# B&R Automation Studio project GAT (part 4)

#### AlarmMgt.st
```iecst
//***********************************************************************
// Copyright: B&R Industrial Automation GmbH
// Author: B&R Industrial Automation GmbH
// Created: Jan 1, 2022
// Description: Tasks for alarm control. The Alarm Management handling is
// done in this task.
//***********************************************************************

PROGRAM _INIT

	// Create folder for this component on the user file device
	DirCreate_New(enable := TRUE, pDevice := ADR('userPartition'), pName := ADR(LOCAL_FOLDER));

	// Check if folder already exist and if so disabled the function block call
	IF DirCreate_New.status = fiERR_DIR_ALREADY_EXIST THEN
		DirCreate_New(enable := FALSE);
	END_IF

	// Initialize mapp function blocks
	MpAlarmXCore_0.Enable := TRUE;
	MpAlarmXCore_0.MpLink := ADR(gMpLinkAlarmXCore);
	MpAlarmXCore_0();

	MpAlarmXHistory_0.Enable := TRUE;
	MpAlarmXHistory_0.DeviceName := ADR('mappAlarmX');
	MpAlarmXHistory_0.MpLink := ADR(gMpLinkAlarmXHistory);
	MpAlarmXHistory_0();

	MpAlarmXListUI_0.Enable := TRUE;
	MpAlarmXListUI_0.UISetup.AlarmListScrollWindow := 10;
	MpAlarmXListUI_0.UISetup.AlarmListSize := 50;
	MpAlarmXListUI_0.UISetup.TimeStampPattern := '%Y %m %d %H:%M:%S';
	MpAlarmXListUI_0();

	MpAlarmXHistoryUI_0.Enable := TRUE;
	MpAlarmXHistoryUI_0.UISetup.AlarmListScrollWindow := 10;
    MpAlarmXHistoryUI_0.UISetup.AlarmListSize := (SIZEOF(MpAlarmXListUIConnect.AlarmList.InstanceID) / SIZEOF(MpAlarmXListUIConnect.AlarmList.InstanceID[0]));
	MpAlarmXHistoryUI_0.UISetup.TimeStampPattern := '%Y %m %d %H:%M:%S';
	MpAlarmXHistoryUI_0();

	// Call action to intialize alarm samples
	AlarmSampleInit;

END_PROGRAM

PROGRAM _CYCLIC

	IF EDGEPOS(SafetyInputs.AcknowledgeAlarms) THEN
        MpAlarmXListUIConnect.AcknowledgeAll := TRUE;
	END_IF

	IF (HmiAlarmX.Commands.ExportAlarms = TRUE) THEN
		MpAlarmXHistory_0.Export := TRUE;
	END_IF

    // Call all cyclic actions
    AlarmHandling;
    GetBacktraceInformation;
    ExecuteQuery;
    QueryTableConfig;
    AlarmSampleFub;

	// Check if any reactions are active.
	// Typically the MpAlarmXCheckReaction() function is called from other tasks within the application.
	// For example, the axis control task might check for the 'Error' reaction to determine whether to send a stop command to the axes.
	// Therefore, copy/paste these IF statements to other places in the application as needed.
    IF MpAlarmXCheckReaction(gMpLinkAlarmXCore, 'Error') THEN
        // Error is active. Add code here to respond to error situation.
    ELSIF MpAlarmXCheckReaction(gMpLinkAlarmXCore, 'Warning') THEN
        // Warning is active. Add code here to respond to warning situation.
	ELSIF MpAlarmXCheckReaction(gMpLinkAlarmXCore, 'Info') THEN
        // Info is active. Add code here to resond to info situation.
	END_IF

	IF ((MpAlarmXHistory_0.Export = TRUE) AND (MpAlarmXHistory_0.CommandDone = TRUE)) THEN
		HmiAlarmX.Commands.ExportAlarms := FALSE;
		MpAlarmXHistory_0.Export := FALSE;
	END_IF

    // Error reset
    IF NOT MpAlarmXCore_0.Error THEN
        MpAlarmXCore_0.ErrorReset := FALSE;
    END_IF
    IF NOT MpAlarmXListUI_0.Error THEN
        MpAlarmXListUI_0.ErrorReset := FALSE;
    END_IF
    IF NOT MpAlarmXHistory_0.Error THEN
        MpAlarmXHistory_0.ErrorReset := FALSE;
    END_IF
    IF NOT MpAlarmXHistoryUI_0.Error THEN
        MpAlarmXHistoryUI_0.ErrorReset := FALSE;
    END_IF

	// Assign MpLinks & UIConnects
	MpAlarmXCore_0.MpLink := ADR(gMpLinkAlarmXCore);
	MpAlarmXListUI_0.MpLink := ADR(gMpLinkAlarmXCore);
	MpAlarmXListUI_0.UIConnect := ADR(MpAlarmXListUIConnect);
	MpAlarmXHistory_0.MpLink := ADR(gMpLinkAlarmXHistory);
	MpAlarmXHistoryUI_0.MpLink := ADR(gMpLinkAlarmXHistory);
	MpAlarmXHistoryUI_0.UIConnect := ADR(MpAlarmXHistoryUIConnect);

	// Call function blocks
	MpAlarmXCore_0();
	MpAlarmXListUI_0();
	MpAlarmXHistory_0();
	MpAlarmXHistoryUI_0();

END_PROGRAM

PROGRAM _EXIT

	// Disable the function blocls to unlink the MpLinks
    MpAlarmXCore_0.Enable := FALSE;
    MpAlarmXListUI_0.Enable := FALSE;
    MpAlarmXHistory_0.Enable := FALSE;
	MpAlarmXHistoryUI_0.Enable := FALSE;
	QueryActiveAlarms.Enable := FALSE;

	// Call function blocks
    MpAlarmXCore_0();
    MpAlarmXListUI_0();
    MpAlarmXHistory_0();
    MpAlarmXHistoryUI_0();
    QueryActiveAlarms();

END_PROGRAM
```

#### AlarmMgt.typ
```iecst
TYPE
	MachineDigitalInputs_type : 	STRUCT  (*Safety related digital inputs of the machine*)
		EmergencyStop : ARRAY[0..MAX_IDX_ESTOP]OF BOOL; (*Emergency stop signal*)
		SafetyDoor : ARRAY[0..MAX_IDX_SAFETY_DOOR]OF BOOL; (*Safety door signal*)
		AcknowledgeAlarms : BOOL;
	END_STRUCT;
	AlarmExamples_typ : 	STRUCT
		LevelMonitoring : INT;
		DeviationMonitoring : INT;
		DeviationMonitoringSetpoint : INT;
		RateOfChange : INT;
		SnippetValue : INT;
		SetControlExample : BOOL;
	END_STRUCT;
	ActiveAlarmState_enum :
		(
		ACTIVE_ALARM_WAIT,
		ACTIVE_ALARM_QUERY,
		ACTIVE_ALARM_NEXT
		);
	AlarmType : 	STRUCT
		Active : BOOL;
		Acknowledged : BOOL;
		Scope : WSTRING[80];
		Name : STRING[80];
		Message : WSTRING[255];
		AdditionalInfo : WSTRING[255];
		TimeStamp : DATE_AND_TIME;
		Code : UDINT;
		Severity : UDINT;
	END_STRUCT;
	AlarmQueryType : 	STRUCT
		Next : BOOL;
		State : ActiveAlarmState_enum;
		LastActiveAlarmUpdateCount : UDINT;
		ActiveAlarmUpdateCount : UDINT;
		Alarms : ARRAY[0..MAX_QUERY_RESULTS]OF AlarmType;
	END_STRUCT;
	AlarmHmiInterface_type : 	STRUCT
		Commands : AlarmCommands_type;
		Status : AlarmStatus_type;
	END_STRUCT;
	AlarmStatus_type : 	STRUCT
		AlarmHistSortCfg : STRING[1000];
		AlarmHistFilterCfg : STRING[1000];
		AlarmSortCfg : STRING[1000];
		AlarmFilterCfg : STRING[1000];
		TableConfig : ARRAY[0..1]OF STRING[120];
	END_STRUCT;
	AlarmCommands_type : 	STRUCT
		ExportAlarms : BOOL;
		RunQuery : BOOL;
	END_STRUCT;
	AlarmQueryHMI_type : 	STRUCT
		Active : ARRAY[0..MAX_QUERY_RESULTS]OF BOOL;
		Acknowledged : ARRAY[0..MAX_QUERY_RESULTS]OF BOOL;
		Scope : ARRAY[0..MAX_QUERY_RESULTS]OF WSTRING[80];
		Name : ARRAY[0..MAX_QUERY_RESULTS]OF STRING[80];
		Message : ARRAY[0..MAX_QUERY_RESULTS]OF WSTRING[255];
		AdditionalInfo : ARRAY[0..MAX_QUERY_RESULTS]OF WSTRING[255];
		TimeStamp : ARRAY[0..MAX_QUERY_RESULTS]OF DATE_AND_TIME;
		Code : ARRAY[0..MAX_QUERY_RESULTS]OF UDINT;
		Severity : ARRAY[0..MAX_QUERY_RESULTS]OF UDINT;
	END_STRUCT;
END_TYPE
```

#### AlarmMgt.var - Local variables
```iecst
(********************************************************************
 * COPYRIGHT -- Bernecker + Rainer
 ********************************************************************
 * Program: FolderHandling
 * File: FolderHandling.var
 * Author: Bernecker + Rainer
 * Created: December , 2020
 ********************************************************************
 * Local variables of program AlarmManagement
 ********************************************************************)
(*Function Blocks--------------------------------------------------------------------------------------------------------------------*)
VAR
	HmiAlarmX : AlarmHmiInterfaceType;
	MpAlarmXHistory_0 : MpAlarmXHistory; (*MpAlarmXHistory instance*)
	MpAlarmXHistoryUI_0 : MpAlarmXHistoryUI; (*MpAlarmXHistoryUI instance*)
	MpAlarmXListUI_0 : MpAlarmXListUI; (*MpAlarmXList instance*)
	MpAlarmXCore_0 : MpAlarmXCore; (*MpAlarmXCore instance*) (*ChangeStyleAlarmButton : USINT := 0; (*changeStyle of a AlarmFlyout in mappView*)
	DirCreate_New : DirCreate;
END_VAR
(*Alarm Management Variables------------------------------------------------------------------------------------------------*)
VAR
	Index : USINT; (*Index to loop through alarm list*)
	MaxIndex : USINT; (*Maximum index for the alarm list*)
	InstanceID : UINT; (*Instance ID*)
	MpAlarmXListUIConnect : MpAlarmXListUIConnectType := (0); (*AlarmVideo : WSTRING[255] := "";
	AlarmInfo : BOOL := 0;*)
	MpAlarmXHistoryUIConnect : MpAlarmXHistoryUIConnectType; (*AlarmX History connection to UI*)
	AlarmQuery : {REDUND_UNREPLICABLE} AlarmQueryType; (*Query Results*)
	QueryActiveAlarms : {REDUND_UNREPLICABLE} MpAlarmXQuery; (*MpAlarmXQuery instance*)
END_VAR
(*Safety Inputs*)
VAR
	SafetyInputs : MachineDigitalInputsType;
END_VAR
(*Defines*)
VAR CONSTANT
	MAX_IDX_ESTOP : UINT := 2;
	MAX_IDX_SAFETY_DOOR : UINT := 5;
	LOCAL_FOLDER : STRING[10] := 'AlarmX';
END_VAR
(*Examples*)
VAR
	CommissioningModeActive : {REDUND_UNREPLICABLE} BOOL; (*Inhibits the Alarms[0] alarm*)
	Alarms : {REDUND_UNREPLICABLE} ARRAY[0..99] OF BOOL; (*Array of active alarm*)
	AlarmExamples : {REDUND_UNREPLICABLE} AlarmExamplesType; (*Sample alarms for different monitoring types*)
	MpAlarmXControlExampleFB : {REDUND_UNREPLICABLE} MpAlarmXAlarmControl; (*MpAlarmXAlarmControl instance*)
END_VAR
VAR CONSTANT
	MAX_QUERY_RESULTS : USINT := 19;
END_VAR
VAR
	AlarmQueryHMI : AlarmQueryHMIType;
	i : USINT;
	EntryCount : USINT;
END_VAR
```

#### AlarmHandling.st
```iecst
ACTION AlarmHandling:

    // CommissioningModeActive = TRUE will inhibit Alarms[0]. The alarm will not trigger even if the alarm condition is active.
	// CommissioningModeActive = FALSE will NOT inhibit Alarms[0]. The alarm will trigger when the alarm condition is active.
	// See Alarm.mpalarmxcore (must enable Advanced Features)
    CommissioningModeActive;

	// Define the condition which triggers each alarm below.
	Alarms[0];

//    Alarms[1] := ;
//    Alarms[2] := ;
//    Alarms[3] := ;
//    Alarms[4] := ;
//    Alarms[5] := ;
//    Alarms[6] := ;
//    Alarms[7] := ;
//    Alarms[8] := ;
//    Alarms[9] := ;
//
//    Alarms[10] := ;
//    Alarms[11] := ;
//    Alarms[12] := ;
//    Alarms[13] := ;
//    Alarms[14] := ;
//    Alarms[15] := ;
//    Alarms[16] := ;
//    Alarms[17] := ;
//    Alarms[18] := ;
//    Alarms[19] := ;
//
//    Alarms[20] := ;
//    Alarms[21] := ;
//    Alarms[22] := ;
//    Alarms[23] := ;
//    Alarms[24] := ;
//    Alarms[25] := ;
//    Alarms[26] := ;
//    Alarms[27] := ;
//    Alarms[28] := ;
//    Alarms[29] := ;
//
//    Alarms[30] := ;
//    Alarms[31] := ;
//    Alarms[32] := ;
//    Alarms[33] := ;
//    Alarms[34] := ;
//    Alarms[35] := ;
//    Alarms[36] := ;
//    Alarms[37] := ;
//    Alarms[38] := ;
//    Alarms[39] := ;
//
//    Alarms[40] := ;
//    Alarms[41] := ;
//    Alarms[42] := ;
//    Alarms[43] := ;
//    Alarms[44] := ;
//    Alarms[45] := ;
//    Alarms[46] := ;
//    Alarms[47] := ;
//    Alarms[48] := ;
//    Alarms[49] := ;
//
//    Alarms[50] := ;
//    Alarms[51] := ;
//    Alarms[52] := ;
//    Alarms[53] := ;
//    Alarms[54] := ;
//    Alarms[55] := ;
//    Alarms[56] := ;
//    Alarms[57] := ;
//    Alarms[58] := ;
//    Alarms[59] := ;
//
//    Alarms[60] := ;
//    Alarms[61] := ;
//    Alarms[62] := ;
//    Alarms[63] := ;
//    Alarms[64] := ;
//    Alarms[65] := ;
//    Alarms[66] := ;
//    Alarms[67] := ;
//    Alarms[68] := ;
//    Alarms[69] := ;
//
//    Alarms[70] := ;
//    Alarms[71] := ;
//    Alarms[72] := ;
//    Alarms[73] := ;
//    Alarms[74] := ;
//    Alarms[75] := ;
//    Alarms[76] := ;
//    Alarms[77] := ;
//    Alarms[78] := ;
//    Alarms[79] := ;
//
//    Alarms[80] := ;
//    Alarms[81] := ;
//    Alarms[82] := ;
//    Alarms[83] := ;
//    Alarms[84] := ;
//    Alarms[85] := ;
//    Alarms[86] := ;
//    Alarms[87] := ;
//    Alarms[88] := ;
//    Alarms[89] := ;
//
//    Alarms[90] := ;
//    Alarms[91] := ;
//    Alarms[92] := ;
//    Alarms[93] := ;
//    Alarms[94] := ;
//    Alarms[95] := ;
//    Alarms[96] := ;
//    Alarms[97] := ;
//    Alarms[98] := ;
//    Alarms[99] := ;

END_ACTION
```

#### HMIActions.st
```iecst
ACTION GetBacktraceInformation:

    MaxIndex := (SIZEOF(MpAlarmXListUIConnect.AlarmList.InstanceID)/SIZEOF(MpAlarmXListUIConnect.AlarmList.InstanceID[0])) - 1;
    // Find selected alarm in order to show backtrace information
    FOR Index := 0 TO MaxIndex DO
        IF (MpAlarmXCore_0.PendingAlarms = 0) THEN
            // No pending alarms, reset instance id
            InstanceID := 0;
            EXIT;
        END_IF

        IF (MpAlarmXListUIConnect.AlarmList.InstanceID[Index] = InstanceID) THEN
            // Found alarm
            MpAlarmXListUIConnect.AlarmList.SelectedIndex := Index;
            EXIT;
        END_IF

        IF (MpAlarmXListUIConnect.AlarmList.InstanceID[Index] = 0) THEN
            IF (MpAlarmXCore_0.PendingAlarms > Index) THEN
                // Alarm not found, List can page up
                MpAlarmXListUIConnect.AlarmList.PageUp := TRUE;
            END_IF
			EXIT;
        ELSIF (Index = MaxIndex) THEN
            // Alarm not found, List can page down
            MpAlarmXListUIConnect.AlarmList.PageDown := TRUE;
        END_IF
	END_FOR

END_ACTION

ACTION QueryTableConfig:

	// Configure visible list
    brsstrcpy(ADR(HmiAlarmX.Status.TableConfig[0]), ADR('{ "specRows": [{"from":'));
    FOR i := 0 TO 9 DO
        IF AlarmQueryHMI.Message[i] <> "" THEN
            EntryCount := i + 1;
        END_IF
    END_FOR
    brsitoa((EntryCount), ADR(HmiAlarmX.Status.TableConfig[0]) + brsstrlen(ADR(HmiAlarmX.Status.TableConfig[0])));
    brsstrcat(ADR(HmiAlarmX.Status.TableConfig[0]),  ADR(',"to":19, "visible":false}]}'));

END_ACTION
```

#### ExecuteQuery.st
```iecst
ACTION ExecuteQuery:

    QueryActiveAlarms.MpLink := ADR(gMpLinkAlarmXCore);
    QueryActiveAlarms.Enable := TRUE;
    QueryActiveAlarms.Name := ADR('ActiveAlarms');
    QueryActiveAlarms.Language := ADR('en');
    QueryActiveAlarms();

    CASE (AlarmQuery.State) OF
        ACTIVE_ALARM_WAIT:
            IF (HmiAlarmX.Commands.RunQuery = TRUE) THEN
                brsmemset(ADR(AlarmQuery.Alarms[0]), 0, SIZEOF(AlarmQuery.Alarms));
                AlarmQuery.LastActiveAlarmUpdateCount := AlarmQuery.ActiveAlarmUpdateCount;
				QueryActiveAlarms.Execute := TRUE;
				HmiAlarmX.Commands.RunQuery := FALSE;
                AlarmQuery.State := ACTIVE_ALARM_QUERY;
            END_IF

        ACTIVE_ALARM_QUERY:
            IF ((QueryActiveAlarms.CommandDone = TRUE) AND (QueryActiveAlarms.Info.HasMoreRows = FALSE)) THEN
                QueryActiveAlarms.Execute := FALSE;
                QueryActiveAlarms.Next := FALSE;
                AlarmQuery.State := ACTIVE_ALARM_WAIT;
            ELSIF ((QueryActiveAlarms.CommandDone = TRUE) AND (QueryActiveAlarms.Info.HasMoreRows = TRUE)) THEN
                QueryActiveAlarms.Next := FALSE;
                AlarmQuery.State := ACTIVE_ALARM_NEXT;
            END_IF

        ACTIVE_ALARM_NEXT:
            IF (AlarmQuery.Next = TRUE) THEN
				// AlarmQuery.Alarms has 20 elements, so it can hold 20 query results at a time.
				// If AlarmQuery.Next is true, this means the query result is more than 20 alarms.
				// If you want to save the data for the first 20 alarms, add code here to copy AlarmQuery.Alarms to another location.
				// Otherwise, the older alarms in the query will get overwritten with the newest entries here.
				brsmemset(ADR(AlarmQuery.Alarms[0]), 0, SIZEOF(AlarmQuery.Alarms));
                AlarmQuery.Next := FALSE;
                QueryActiveAlarms.Next := TRUE;
                AlarmQuery.State := ACTIVE_ALARM_QUERY;
            END_IF
	END_CASE

	// Convert the query results into arrays that can easily be bound to the Table widget in mapp View
	FOR i:=0 TO MAX_QUERY_RESULTS DO
		AlarmQueryHMI.Active[i] := AlarmQuery.Alarms[i].Active;
		AlarmQueryHMI.Acknowledged[i] := AlarmQuery.Alarms[i].Acknowledged;
		AlarmQueryHMI.Scope[i] := AlarmQuery.Alarms[i].Scope;
		AlarmQueryHMI.Name[i] := AlarmQuery.Alarms[i].Name;
		AlarmQueryHMI.Message[i] := AlarmQuery.Alarms[i].Message;
		AlarmQueryHMI.AdditionalInfo[i] := AlarmQuery.Alarms[i].AdditionalInfo;
		AlarmQueryHMI.TimeStamp[i] := AlarmQuery.Alarms[i].TimeStamp;
		AlarmQueryHMI.Severity[i] := AlarmQuery.Alarms[i].Severity;
	END_FOR

END_ACTION
```

#### AlarmSamples.st
```iecst
ACTION AlarmSampleInit:

    // Call all variables that are needed for the alarm examples and explain all examples in comments

    // If AlarmExamples.LevelMonitoring gets less than 20 or more than 80, the LevelMonitoringExample alarm will trigger
	// The Low limit is 20. The LowLow limit is 10. The High limit is 80. The HighHigh limit is 90.
	AlarmExamples.LevelMonitoring := 50;

	// If AlarmExamples.DeviationMonitoring deviates from the setpoint (AlarmExamples.DeviationMonitoringSetpoint) by more than 5
	// units in either direction, the DeviationMonitoringExample alarm will trigger
	AlarmExamples.DeviationMonitoring := 15;
	AlarmExamples.DeviationMonitoringSetpoint := 15;

	// If AlarmExamples.RateOfChange increases at a rate of more than 5 units per second, the RateOfChangeExample alarm will trigger
	AlarmExamples.RateOfChange := 0;

	//If AlarmExamples.SnippetValue gets between 50 and 100, an alarm will trigger and the current value will be shown in the alarm text
	AlarmExamples.SnippetValue := 10;

END_ACTION

ACTION AlarmSampleFub:

	// Example of using the MpAlarmXControl() function block.
	// Typically this function is called from other tasks within the application (decentralized).
	// For example, if you have an error in the recipe system, you can trigger it directly in the recipe task.
	// Therefore, copy/paste this example to other places in the application as needed.

	MpAlarmXControlExampleFB.MpLink := ADR(gMpLinkAlarmXCore);
	MpAlarmXControlExampleFB.Enable := TRUE;
	MpAlarmXControlExampleFB.Name := ADR('MpAlarmXControlExample');
	MpAlarmXControlExampleFB.Set := AlarmExamples.SetControlExample;
	MpAlarmXControlExampleFB();

END_ACTION
```

### Program Logical/Infrastructure/AlarmX/AlarmX

#### AlarmSamples.st
```iecst
ACTION AlarmSampleInit:

    // Call all variables that are needed for the alarm examples and explain all examples in comments

    // If AlarmExamples.LevelMonitoring gets less than 20 or more than 80, the LevelMonitoringExample alarm will trigger
	// The Low limit is 20. The LowLow limit is 10. The High limit is 80. The HighHigh limit is 90.
    AlarmExamples.LevelMonitoring := 50;

	// If AlarmExamples.DeviationMonitoring deviates from the setpoint (AlarmExamples.DeviationMonitoringSetpoint) by more than 5
	// units in either direction, the DeviationMonitoringExample alarm will trigger
	AlarmExamples.DeviationMonitoring := 15;
	AlarmExamples.DeviationMonitoringSetpoint := 15;

	// If AlarmExamples.RateOfChange increases at a rate of more than 5 units per second, the RateOfChangeExample alarm will trigger
	AlarmExamples.RateOfChange := 0;

	//If AlarmExamples.SnippetValue gets between 50 and 100, an alarm will trigger and the current value will be shown in the alarm text
	AlarmExamples.SnippetValue := 10;

END_ACTION

ACTION AlarmSampleFub:

	// Example of using the MpAlarmXControl() function block.
	// Typically this function is called from other tasks within the application (decentralized).
	// For example, if you have an error in the recipe system, you can trigger it directly in the recipe task.
	// Therefore, copy/paste this example to other places in the application as needed.
    MpAlarmXControlExampleFB.MpLink := ADR(gMpLinkAlarmXCore);
    MpAlarmXControlExampleFB.Enable := TRUE;
    MpAlarmXControlExampleFB.Name := ADR('MpAlarmXControlExample');
    MpAlarmXControlExampleFB.Set := AlarmExamples.SetControlExample;
    MpAlarmXControlExampleFB();

END_ACTION
```

### Package Logical/Infrastructure/Audit - Package for mapp Audit Framework

### Program Logical/Infrastructure/Audit/AuditMgr (IEC) - Audit manager

#### AuditMgt.st - Init, cyclic, exit code
```iecst
//*********************************************************************************
//* Copyright: B&R Industrial Automation GmbH
//* Author:    B&R Industrial Automation GmbH
//* Created:   30. Dec 2020/08:00
//* Description: Tasks FOR Audit Management.  The Audit Management is done in this task.
//********************************************************************************

PROGRAM _INIT

	//Create folder for this component on the user file device
	DirCreate_New(enable := TRUE, pDevice := ADR('userPartition'), pName := ADR(LOCAL_FOLDER));

	//Check if folder already exist and if so disabled the function block call
	IF DirCreate_New.status = fiERR_DIR_ALREADY_EXIST THEN
		DirCreate_New(enable := FALSE);
	END_IF

	// Init function blocks
	MpAuditTrail_0.MpLink := ADR(gAuditTrailMpLink);
	MpAuditTrail_0.Enable := TRUE;
	MpAuditTrail_0.DeviceName := ADR('mappAuditFiles');

	MpFileManagerUI_0.Enable := TRUE;
	MpFileManagerUI_0.MpLink := ADR(gMpLinkFileManagerUIAudit);
	MpFileManagerUI_0.UIConnect := ADR(MpFileManagerUIConnect);
	MpFileManagerUI_0.UISetup.FileListSize := 50;

	// Filter files for pdf type
	MpFileManagerUIConnect.File.Filter := '*.pdf';
END_PROGRAM

PROGRAM _CYCLIC
	// Reset export command
	IF MpAuditTrail_0.CommandDone THEN
		MpAuditTrail_0.Export := FALSE;
		MpFileManagerUIConnect.File.Refresh := TRUE;
	END_IF

	// Reset error reset
	IF NOT MpAuditTrail_0.Error THEN
	  MpAuditTrail_0.ErrorReset := FALSE;
	END_IF

    // Save Filenames to a seperate array for display in Table
	FOR i := 0 TO 49 DO
        DisplayFileName[i] := MpFileManagerUIConnect.File.List.Items[i].Name;
        // if selected set a index for display selected file in table
		IF DisplayFileNameIndex = INT_TO_USINT(i) THEN
			MpFileManagerUIConnect.File.List.Items[i].IsSelected := TRUE;
		END_IF
    END_FOR

    // String for pdfViewer to display right report
	StrSelectedFile := CONCAT(STR_FILE_DEVICE, MpFileManagerUIConnect.File.List.Items[DisplayFileNameIndex].Name);

	// Configure visible file list
	brsstrcpy(ADR(TableConfig), ADR('{ "specRows": [{"from":'));
	brsitoa(MpFileManagerUIConnect.File.PathInfo.FileCount, ADR(TableConfig) + brsstrlen(ADR(TableConfig)));
	brsstrcat(ADR(TableConfig),  ADR(',"to":49, "visible":false}]}'));

	// Call function blocks
	MpAuditTrail_0();
	MpFileManagerUI_0();
END_PROGRAM

PROGRAM _EXIT
	// Insert code here

END_PROGRAM
```

#### AuditMgr.var - not listed in the package file held
```iecst
(********************************************************************
 * COPYRIGHT -- Bernecker + Rainer
 ********************************************************************
 * Program: FolderHandling
 * File: FolderHandling.var
 * Author: Bernecker + Rainer
 * Created: December , 2020
 ********************************************************************
 * Local variables of program Audit Management
 ********************************************************************)
(*Audit Management Related Function Blocks*)
VAR
	MpAuditTrail_0 : MpAuditTrail; (*mapp Audit function block*)
	MpFileManagerUIConnect : MpFileManagerUIConnectType := (DeviceList:=(DeviceNames:=['mappAuditFiles',9('')])); (*mapp File Manager to UI Connect*)
	MpFileManagerUI_0 : MpFileManagerUI;
	DirCreate_0 : DirCreate;
END_VAR
(*Audit Management Related Variables*)
VAR
	TableConfig : STRING[80];
	i : INT;
	DisplayFileNameIndex : USINT := 0; (*index of selected file for display in table in mappView*)
	StrSelectedFile : STRING[256] := '0'; (*Gives the path of selected report to pdfViewer in mappView*)
	DisplayFileName : ARRAY[0..49] OF STRING[255] := [50('')]; (*Displayed Files for mappView*)
	STR_FILE_DEVICE : STRING[80] := '/FileDevice:mappAudit/'; (*File Device*)
END_VAR
VAR CONSTANT
	LOCAL_FOLDER : STRING[10] := 'Audit';
END_VAR
```

#### AuditMgr.st - not listed in the package file held
```iecst
//*********************************************************************************
//* Copyright: B&R Industrial Automation GmbH
//* Author:    B&R Industrial Automation GmbH
//* Created:   30. Dec 2020/08:00
//* Description: Tasks FOR Audit Management.  The Audit Management is done in this task.
//********************************************************************************

PROGRAM _INIT

	// Create folder for this component on the user file device
	DirCreate_0(enable := TRUE, pDevice := ADR('UserPartition'), pName := ADR(LOCAL_FOLDER));

	// Check if folder already exist and if so disabled the function block call
	IF DirCreate_0.status = fiERR_DIR_ALREADY_EXIST THEN
		DirCreate_0(enable := FALSE);
	END_IF

	// Init function blocks
	MpAuditTrail_0.MpLink := ADR(gAuditTrailMpLink);
	MpAuditTrail_0.Enable := TRUE;
	MpAuditTrail_0.DeviceName := ADR('mappAuditFiles');

	MpFileManagerUI_0.Enable := TRUE;
	MpFileManagerUI_0.MpLink := ADR(gMpLinkFileManagerUIAudit);
	MpFileManagerUI_0.UIConnect := ADR(MpFileManagerUIConnect);
	MpFileManagerUI_0.UISetup.FileListSize := 50;

	// Filter files for pdf type
	MpFileManagerUIConnect.File.Filter := '*.pdf';
END_PROGRAM

PROGRAM _CYCLIC
	// Reset export command
	IF MpAuditTrail_0.CommandDone THEN
		MpAuditTrail_0.Export := FALSE;
		MpFileManagerUIConnect.File.Refresh := TRUE;
	END_IF

	// Reset error reset
	IF NOT MpAuditTrail_0.Error THEN
	  MpAuditTrail_0.ErrorReset := FALSE;
	END_IF

    // Save Filenames to a seperate array for display in Table
	FOR i := 0 TO 49 DO
        DisplayFileName[i] := MpFileManagerUIConnect.File.List.Items[i].Name;
        // If selected set a index for display selected file in table
		IF DisplayFileNameIndex = INT_TO_USINT(i) THEN
			MpFileManagerUIConnect.File.List.Items[i].IsSelected := TRUE;
		END_IF
    END_FOR

    // String for pdfViewer to display right report
	StrSelectedFile := CONCAT(STR_FILE_DEVICE, MpFileManagerUIConnect.File.List.Items[DisplayFileNameIndex].Name);

	// Configure visible file list
	brsstrcpy(ADR(TableConfig), ADR('{ "specRows": [{"from":'));
	brsitoa(MpFileManagerUIConnect.File.PathInfo.FileCount, ADR(TableConfig) + brsstrlen(ADR(TableConfig)));
	brsstrcat(ADR(TableConfig),  ADR(',"to":49, "visible":false}]}'));

	// Call function blocks
	MpAuditTrail_0();
	MpFileManagerUI_0();
END_PROGRAM

PROGRAM _EXIT
	// Insert code here

END_PROGRAM
```

### Program Logical/Infrastructure/Audit/AuditMgt

#### AuditMgt.var
```iecst
(********************************************************************
 * COPYRIGHT -- Bernecker + Rainer
 ********************************************************************
 * Program: FolderHandling
 * File: FolderHandling.var
 * Author: Bernecker + Rainer
 * Created: December , 2020
 ********************************************************************
 * Local variables of program Audit Management
 ********************************************************************)
(*Audit Management Related Function Blocks*)
VAR
	MpAuditTrail_0 : MpAuditTrail; (*mapp Audit function block*)
	MpFileManagerUIConnect : MpFileManagerUIConnectType := (DeviceList:=(DeviceNames:=['mappAuditFiles',9('')])); (*mapp File Manager to UI Connect*)
	MpFileManagerUI_0 : MpFileManagerUI;
	DirCreate_New : DirCreate;
END_VAR
(*Audit Management Related Variables*)
VAR
	TableConfig : STRING[80];
	i : INT;
	DisplayFileNameIndex : USINT := 0; (*index of selected file for display in table in mappView*)
	StrSelectedFile : STRING[256] := '0'; (*Gives the path of selected report to pdfViewer in mappView*)
	DisplayFileName : ARRAY[0..49] OF STRING[255] := [50('')]; (*Displayed Files for mappView*)
	STR_FILE_DEVICE : STRING[80] := '/FileDevice:mappAudit/'; (*File Device*)
END_VAR
VAR CONSTANT
	LOCAL_FOLDER : STRING[10] := 'Audit';
END_VAR
```

#### AuditMgt.st
```iecst
//*********************************************************************************
//* Copyright: B&R Industrial Automation GmbH
//* Author:    B&R Industrial Automation GmbH
//* Created:   30. Dec 2020/08:00
//* Description: Tasks FOR Audit Management.  The Audit Management is done in this task.
//********************************************************************************

PROGRAM _INIT

	//Create folder for this component on the user file device
	DirCreate_New(enable := TRUE, pDevice := ADR('userPartition'), pName := ADR(LOCAL_FOLDER));

	//Check if folder already exist and if so disabled the function block call
	IF DirCreate_New.status = fiERR_DIR_ALREADY_EXIST THEN
		DirCreate_New(enable := FALSE);
	END_IF

	// Init function blocks
	MpAuditTrail_0.MpLink := ADR(gAuditTrailMpLink);
	MpAuditTrail_0.Enable := TRUE;
	MpAuditTrail_0.DeviceName := ADR('mappAudit');

	MpFileManagerUI_0.Enable := TRUE;
	MpFileManagerUI_0.MpLink := ADR(gMpLinkFileManagerUIAudit);
	MpFileManagerUI_0.UIConnect := ADR(MpFileManagerUIConnect);
	MpFileManagerUI_0.UISetup.FileListSize := 50;

	// Filter files for pdf type
	MpFileManagerUIConnect.File.Filter := '*.pdf';
END_PROGRAM

PROGRAM _CYCLIC
	// Reset export command
	IF MpAuditTrail_0.CommandDone THEN
		MpAuditTrail_0.Export := FALSE;
		MpFileManagerUIConnect.File.Refresh := TRUE;
	END_IF

	// Reset error reset
	IF NOT MpAuditTrail_0.Error THEN
	  MpAuditTrail_0.ErrorReset := FALSE;
	END_IF

    // Save Filenames to a seperate array for display in Table
	FOR i := 0 TO 49 DO
        DisplayFileName[i] := MpFileManagerUIConnect.File.List.Items[i].Name;
        // if selected set a index for display selected file in table
		IF DisplayFileNameIndex = INT_TO_USINT(i) THEN
			MpFileManagerUIConnect.File.List.Items[i].IsSelected := TRUE;
		END_IF
    END_FOR

    // String for pdfViewer to display right report
	StrSelectedFile := CONCAT(STR_FILE_DEVICE, MpFileManagerUIConnect.File.List.Items[DisplayFileNameIndex].Name);

	// Configure visible file list
	brsstrcpy(ADR(TableConfig), ADR('{ "specRows": [{"from":'));
	brsitoa(MpFileManagerUIConnect.File.PathInfo.FileCount, ADR(TableConfig) + brsstrlen(ADR(TableConfig)));
	brsstrcat(ADR(TableConfig),  ADR(',"to":49, "visible":false}]}'));

	// Call function blocks
	MpAuditTrail_0();
	MpFileManagerUI_0();
END_PROGRAM

PROGRAM _EXIT
	// Insert code here

END_PROGRAM
```

### Package Logical/Infrastructure/Data - Package for mapp Data Framework

### Program Logical/Infrastructure/Data/DataMgr (IEC) - Data manager

#### DataMgr.st - Init, cyclic, exit code
```iecst
//*********************************************************************************
//* Copyright: B&R Industrial Automation GmbH
//* Author:    B&R Industrial Automation GmbH
//* Created:   30. Sep 2020/08:00
//* Description: Tasks FOR Data Management control. The Data Management handling is done in this task.
//*********************************************************************************

PROGRAM _INIT

	// Create folder for this component on the user file device
	DirCreate_New(enable := TRUE, pDevice := ADR('UserPartition'), pName := ADR(LOCAL_FOLDER));

	// Check if folder already exist and if so disabled the function block call
	IF DirCreate_New.status = fiERR_DIR_ALREADY_EXIST THEN
		DirCreate_New(enable := FALSE);
	END_IF

	// Init mapp function blocks
	MpFileManagerUI_0.Enable := TRUE;
	MpFileManagerUI_0.MpLink := ADR(gMpLinkFileManagerUIData);
	MpFileManagerUI_0.UIConnect := ADR(MpFileManagerUIConnect);

	MpDataRecorder_0.MpLink := ADR(gMpLinkDataRecorder);
	MpDataRecorder_0.Enable := TRUE ;
	MpDataRecorder_0.DeviceName := ADR('mappDataFiles');
	MpDataRecorder_0.RecordMode := mpDATA_RECORD_MODE_TIME;
	MpDataRecorder_0.SamplingTime := t#5s;

	// Register PVs for data recording
	MpDataRegPar_x[0].MpLink := ADR(gMpLinkDataRecorder);
	MpDataRegPar_x[0].Enable := TRUE;
	MpDataRegPar_x[0].PVName := ADR('PIDControl:rActValue');
	MpDataRegPar_x[0].Description := ADR('Control Value');

	MpDataRegPar_x[1].MpLink := ADR(gMpLinkDataRecorder);
	MpDataRegPar_x[1].Enable := TRUE;
	MpDataRegPar_x[1].PVName := ADR('MainCtrl:MpAxisBasic_x[0].Velocity');
	MpDataRegPar_x[1].Description := ADR('Feeder Velocity');

	// Filter files for pdf type
	MpFileManagerUIConnect.File.Filter := '*.pdf';
END_PROGRAM

PROGRAM _CYCLIC
	//***************************************************
	FOR i := 0 TO 49 DO
		// Save Filenames to a seperate array for display in Table
		DisplayFileName[i] := MpFileManagerUIConnect.File.List.Items[i].Name;
		// Mark file selection
		MpFileManagerUIConnect.File.List.Items[i].IsSelected := (DisplayFileNameIndex = INT_TO_USINT(i));
    END_FOR
    // String for pdfViewer to display right report
	StrSelectedFile := CONCAT(STR_FILE_DEVICE, MpFileManagerUIConnect.File.List.Items[DisplayFileNameIndex].Name);

	// Configure visible file list
	brsstrcpy(ADR(TableConfig), ADR('{ "specRows": [{"from":'));
	brsitoa(MpFileManagerUIConnect.File.PathInfo.FileCount, ADR(TableConfig) + brsstrlen(ADR(TableConfig)));
	brsstrcat(ADR(TableConfig),  ADR(',"to":49, "visible":false}]}'));

	// Call function blocks
	MpDataRecorder_0();
	FOR i := 0 TO MAX_IDX_DATA_REG DO
		MpDataRegPar_x[i]();
	END_FOR
	MpFileManagerUI_0();

	// Reset ErrorReset command
	IF NOT MpDataRecorder_0.Error THEN
		MpDataRecorder_0.ErrorReset := FALSE;
	END_IF
	FOR i := 0 TO MAX_IDX_DATA_REG DO
		IF NOT MpDataRegPar_x[i].Error THEN
			MpDataRegPar_x[i].ErrorReset := FALSE;
		END_IF
	END_FOR
END_PROGRAM

PROGRAM _EXIT
	// Call mapp function blocks with enable = false
	MpFileManagerUI_0.Enable := FALSE;
	MpFileManagerUI_0();
	MpDataRecorder_0.Enable := FALSE;
	MpDataRecorder_0();
	FOR i := 0 TO MAX_IDX_DATA_REG DO
		MpDataRegPar_x[i].Enable := FALSE;
		MpDataRegPar_x[i]();
	END_FOR
END_PROGRAM
```

#### DataMgr.var - Local variables
```iecst
(********************************************************************
 * COPYRIGHT -- Bernecker + Rainer
 ********************************************************************
 * Program: FolderHandling
 * File: FolderHandling.var
 * Author: Bernecker + Rainer
 * Created: December , 2020
 ********************************************************************
 * Local variables of program Data Management
 ********************************************************************)
(*Data Management Related Variables*)
VAR
	i : INT; (*index used in for loop*)
	MpDataRecorder_0 : MpDataRecorder; (*mapp Data Recorder Function block*)
	MpDataRegPar_x : ARRAY[0..MAX_IDX_DATA_REG] OF MpDataRegPar; (*Function Block to Set the recorded variable*)
	MpFileManagerUIConnect : MpFileManagerUIConnectType := (DeviceList:=(DeviceNames:=['mappDataFiles',9('')]));
	DirCreate_0 : DirCreate;
END_VAR
(*Data Management Related Function Blocks*)
VAR
	MpFileManagerUI_0 : MpFileManagerUI; (*File Manager Function Block*)
	DisplayFileName : ARRAY[0..49] OF STRING[80]; (*Displayed File Name*)
	StrSelectedFile : STRING[80]; (*Selected File*)
	TableConfig : STRING[80];
	DisplayFileNameIndex : USINT; (*Selected file index*)
END_VAR
(*Constants*)
VAR CONSTANT
	MAX_IDX_DATA_REG : USINT := 1; (*Max index of registered variables for MpData*)
	STR_FILE_DEVICE : STRING[256] := '/FileDevice:mappData/'; (*File Device for mappData*)
	LOCAL_FOLDER : STRING[10] := 'Data';
END_VAR
```

#### DataMgt.var - not listed in the package file held
```iecst
(********************************************************************
 * COPYRIGHT -- Bernecker + Rainer
 ********************************************************************
 * Program: FolderHandling
 * File: FolderHandling.var
 * Author: Bernecker + Rainer
 * Created: December , 2020
 ********************************************************************
 * Local variables of program Data Management
 ********************************************************************)
(*Data Management Related Variables*)
VAR
	i : INT; (*index used in for loop*)
	MpDataRecorder_0 : MpDataRecorder; (*mapp Data Recorder Function block*)
	MpDataRegPar_x : ARRAY[0..MAX_IDX_DATA_REG] OF MpDataRegPar; (*Function Block to Set the recorded variable*)
	MpFileManagerUIConnect : MpFileManagerUIConnectType := (DeviceList:=(DeviceNames:=['mappDataFiles',9('')]));
	DirCreate_New : DirCreate;
END_VAR
(*Data Management Related Function Blocks*)
VAR
	MpFileManagerUI_0 : MpFileManagerUI; (*File Manager Function Block*)
	DisplayFileName : ARRAY[0..49] OF STRING[80]; (*Displayed File Name*)
	StrSelectedFile : STRING[80]; (*Selected File*)
	TableConfig : STRING[80];
	DisplayFileNameIndex : USINT; (*Selected file index*)
END_VAR
(*Constants*)
VAR CONSTANT
	MAX_IDX_DATA_REG : USINT := 1; (*Max index of registered variables for MpData*)
	STR_FILE_DEVICE : STRING[256] := '/FileDevice:mappData/'; (*File Device for mappData*)
	LOCAL_FOLDER : STRING[10] := 'Data';
END_VAR
```

#### DataMgt.st - not listed in the package file held
```iecst
//*********************************************************************************
//* Copyright: B&R Industrial Automation GmbH
//* Author:    B&R Industrial Automation GmbH
//* Created:   30. Sep 2020/08:00
//* Description: Tasks FOR Data Management control. The Data Management handling is done in this task.
//*********************************************************************************

PROGRAM _INIT

	//Create folder for this component on the user file device
	DirCreate_New(enable := TRUE, pDevice := ADR('userPartition'), pName := ADR(LOCAL_FOLDER));

	//Check if folder already exist and if so disabled the function block call
	IF DirCreate_New.status = fiERR_DIR_ALREADY_EXIST THEN
		DirCreate_New(enable := FALSE);
	END_IF

	// Init mapp function blocks
	MpFileManagerUI_0.Enable := TRUE;
	MpFileManagerUI_0.MpLink := ADR(gMpLinkFileManagerUIData);
	MpFileManagerUI_0.UIConnect := ADR(MpFileManagerUIConnect);

	MpDataRecorder_0.MpLink := ADR(gMpLinkDataRecorder);
	MpDataRecorder_0.Enable := TRUE ;
	MpDataRecorder_0.DeviceName := ADR('mappDataFiles');
	MpDataRecorder_0.RecordMode := mpDATA_RECORD_MODE_TIME;
	MpDataRecorder_0.SamplingTime := t#5s;

	// Register PVs for data recording
	MpDataRegPar_x[0].MpLink := ADR(gMpLinkDataRecorder);
	MpDataRegPar_x[0].Enable := TRUE;
	MpDataRegPar_x[0].PVName := ADR('PIDControl:rActValue');
	MpDataRegPar_x[0].Description := ADR('Control Value');

	MpDataRegPar_x[1].MpLink := ADR(gMpLinkDataRecorder);
	MpDataRegPar_x[1].Enable := TRUE;
	MpDataRegPar_x[1].PVName := ADR('MainCtrl:MpAxisBasic_x[0].Velocity');
	MpDataRegPar_x[1].Description := ADR('Feeder Velocity');

	// Filter files for pdf type
	MpFileManagerUIConnect.File.Filter := '*.pdf';
END_PROGRAM

PROGRAM _CYCLIC
	//***************************************************
	FOR i := 0 TO 49 DO
		// Save Filenames to a seperate array for display in Table
		DisplayFileName[i] := MpFileManagerUIConnect.File.List.Items[i].Name;
		// mark file selection
		MpFileManagerUIConnect.File.List.Items[i].IsSelected := (DisplayFileNameIndex = INT_TO_USINT(i));
    END_FOR
    // String for pdfViewer to display right report
	StrSelectedFile := CONCAT(STR_FILE_DEVICE, MpFileManagerUIConnect.File.List.Items[DisplayFileNameIndex].Name);

	// Configure visible file list
	brsstrcpy(ADR(TableConfig), ADR('{ "specRows": [{"from":'));
	brsitoa(MpFileManagerUIConnect.File.PathInfo.FileCount, ADR(TableConfig) + brsstrlen(ADR(TableConfig)));
	brsstrcat(ADR(TableConfig),  ADR(',"to":49, "visible":false}]}'));

	// Call function blocks
	MpDataRecorder_0();
	FOR i := 0 TO MAX_IDX_DATA_REG DO
		MpDataRegPar_x[i]();
	END_FOR
	MpFileManagerUI_0();

	// Reset ErrorReset command
	IF NOT MpDataRecorder_0.Error THEN
		MpDataRecorder_0.ErrorReset := FALSE;
	END_IF
	FOR i := 0 TO MAX_IDX_DATA_REG DO
		IF NOT MpDataRegPar_x[i].Error THEN
			MpDataRegPar_x[i].ErrorReset := FALSE;
		END_IF
	END_FOR
END_PROGRAM

PROGRAM _EXIT
	// call mapp function blocks with enable = false
	MpFileManagerUI_0.Enable := FALSE;
	MpFileManagerUI_0();
	MpDataRecorder_0.Enable := FALSE;
	MpDataRecorder_0();
	FOR i := 0 TO MAX_IDX_DATA_REG DO
		MpDataRegPar_x[i].Enable := FALSE;
		MpDataRegPar_x[i]();
	END_FOR
END_PROGRAM
```

### Program Logical/Infrastructure/Data/DataMgt (IEC)

#### DataMgt.st - Init, cyclic, exit code
```iecst
//*********************************************************************************
//* Copyright: B&R Industrial Automation GmbH
//* Author:    B&R Industrial Automation GmbH
//* Created:   30. Sep 2020/08:00
//* Description: Tasks FOR Data Management control. The Data Management handling is done in this task.
//*********************************************************************************

PROGRAM _INIT

	//Create folder for this component on the user file device
	DirCreate_New(enable := TRUE, pDevice := ADR('userPartition'), pName := ADR(LOCAL_FOLDER));

	//Check if folder already exist and if so disabled the function block call
	IF DirCreate_New.status = fiERR_DIR_ALREADY_EXIST THEN
		DirCreate_New(enable := FALSE);
	END_IF

	// Init mapp function blocks
	MpFileManagerUI_0.Enable := TRUE;
	MpFileManagerUI_0.MpLink := ADR(gMpLinkFileManagerUIData);
	MpFileManagerUI_0.UIConnect := ADR(MpFileManagerUIConnect);

	MpDataRecorder_0.MpLink := ADR(gMpLinkDataRecorder);
	MpDataRecorder_0.Enable := TRUE ;
	MpDataRecorder_0.DeviceName := ADR('mappData');
	MpDataRecorder_0.RecordMode := mpDATA_RECORD_MODE_TIME;
	MpDataRecorder_0.SamplingTime := t#5s;

	// Register PVs for data recording
	MpDataRegPar_x[0].MpLink := ADR(gMpLinkDataRecorder);
	MpDataRegPar_x[0].Enable := TRUE;
	MpDataRegPar_x[0].PVName := ADR('PIDControl:rActValue');
	MpDataRegPar_x[0].Description := ADR('Control Value');

	MpDataRegPar_x[1].MpLink := ADR(gMpLinkDataRecorder);
	MpDataRegPar_x[1].Enable := TRUE;
	MpDataRegPar_x[1].PVName := ADR('MainCtrl:MpAxisBasic_x[0].Velocity');
	MpDataRegPar_x[1].Description := ADR('Feeder Velocity');

	// Filter files for pdf type
	MpFileManagerUIConnect.File.Filter := '*.pdf';
END_PROGRAM

PROGRAM _CYCLIC
	//***************************************************
	FOR i := 0 TO 49 DO
		// Save Filenames to a seperate array for display in Table
		DisplayFileName[i] := MpFileManagerUIConnect.File.List.Items[i].Name;
		// mark file selection
		MpFileManagerUIConnect.File.List.Items[i].IsSelected := (DisplayFileNameIndex = INT_TO_USINT(i));
    END_FOR
    // String for pdfViewer to display right report
	StrSelectedFile := CONCAT(STR_FILE_DEVICE, MpFileManagerUIConnect.File.List.Items[DisplayFileNameIndex].Name);

	// Configure visible file list
	brsstrcpy(ADR(TableConfig), ADR('{ "specRows": [{"from":'));
	brsitoa(MpFileManagerUIConnect.File.PathInfo.FileCount, ADR(TableConfig) + brsstrlen(ADR(TableConfig)));
	brsstrcat(ADR(TableConfig),  ADR(',"to":49, "visible":false}]}'));

	// Call function blocks
	MpDataRecorder_0();
	FOR i := 0 TO MAX_IDX_DATA_REG DO
		MpDataRegPar_x[i]();
	END_FOR
	MpFileManagerUI_0();

	// Reset ErrorReset command
	IF NOT MpDataRecorder_0.Error THEN
		MpDataRecorder_0.ErrorReset := FALSE;
	END_IF
	FOR i := 0 TO MAX_IDX_DATA_REG DO
		IF NOT MpDataRegPar_x[i].Error THEN
			MpDataRegPar_x[i].ErrorReset := FALSE;
		END_IF
	END_FOR
END_PROGRAM

PROGRAM _EXIT
	// call mapp function blocks with enable = false
	MpFileManagerUI_0.Enable := FALSE;
	MpFileManagerUI_0();
	MpDataRecorder_0.Enable := FALSE;
	MpDataRecorder_0();
	FOR i := 0 TO MAX_IDX_DATA_REG DO
		MpDataRegPar_x[i].Enable := FALSE;
		MpDataRegPar_x[i]();
	END_FOR
END_PROGRAM
```

#### DataMgt.var - Local variables
```iecst
(********************************************************************
 * COPYRIGHT -- Bernecker + Rainer
 ********************************************************************
 * Program: FolderHandling
 * File: FolderHandling.var
 * Author: Bernecker + Rainer
 * Created: December , 2020
 ********************************************************************
 * Local variables of program Data Management
 ********************************************************************)
(*Data Management Related Variables*)
VAR
	i : INT; (*index used in for loop*)
	MpDataRecorder_0 : MpDataRecorder; (*mapp Data Recorder Function block*)
	MpDataRegPar_x : ARRAY[0..MAX_IDX_DATA_REG] OF MpDataRegPar; (*Function Block to Set the recorded variable*)
	MpFileManagerUIConnect : MpFileManagerUIConnectType := (DeviceList:=(DeviceNames:=['mappData',9('')]));
	DirCreate_New : DirCreate;
END_VAR
(*Data Management Related Function Blocks*)
VAR
	MpFileManagerUI_0 : MpFileManagerUI; (*File Manager Function Block*)
	DisplayFileName : ARRAY[0..49] OF STRING[80]; (*Displayed File Name*)
	StrSelectedFile : STRING[80]; (*Selected File*)
	TableConfig : STRING[80];
	DisplayFileNameIndex : USINT; (*Selected file index*)
END_VAR
(*Constants*)
VAR CONSTANT
	MAX_IDX_DATA_REG : USINT := 1; (*Max index of registered variables for MpData*)
	STR_FILE_DEVICE : STRING[256] := '/FileDevice:mappData/'; (*File Device for mappData*)
	LOCAL_FOLDER : STRING[10] := 'Data';
END_VAR
```

#### DataMgtst.st - not listed in the package file held
```iecst
(*********************************************************************************
* Copyright: B&R Industrial Automation GmbH
* Author:    B&R Industrial Automation GmbH
* Created:   30. Sep 2020/08:00
* Description: Tasks FOR Data Management control. The Data Management handling is done in this task.
*********************************************************************************)

PROGRAM _INIT

	(*Create folder for this component on the user file device*)
	DirCreate_New(enable := TRUE, pDevice := ADR('userPartition'), pName := ADR(LOCAL_FOLDER));

	(*Check if folder already exist and if so disabled the function block call*)
	IF DirCreate_New.status = fiERR_DIR_ALREADY_EXIST THEN
		DirCreate_New(enable := FALSE);
	END_IF

	(* Init mapp function blocks *)
	MpFileManagerUI_0.Enable			:= TRUE;
	MpFileManagerUI_0.MpLink			:= ADR(gMpLinkFileManagerUIData);
	MpFileManagerUI_0.UIConnect			:= ADR(MpFileManagerUIConnect);

	MpDataRecorder_0.MpLink				:= ADR(gMpLinkDataRecorder);
	MpDataRecorder_0.Enable				:= TRUE ;
	MpDataRecorder_0.DeviceName			:= ADR('mappData');
	MpDataRecorder_0.RecordMode			:= mpDATA_RECORD_MODE_TIME;
	MpDataRecorder_0.SamplingTime		:= t#5s;

	(* Register PVs for data recording *)
	MpDataRegPar_x[0].MpLink			:= ADR(gMpLinkDataRecorder);
	MpDataRegPar_x[0].Enable			:= TRUE;
	MpDataRegPar_x[0].PVName			:= ADR('PIDControl:rActValue');
	MpDataRegPar_x[0].Description		:= ADR('Control Value');

	MpDataRegPar_x[1].MpLink			:= ADR(gMpLinkDataRecorder);
	MpDataRegPar_x[1].Enable			:= TRUE;
	MpDataRegPar_x[1].PVName			:= ADR('MainCtrl:MpAxisBasic_x[0].Velocity');
	MpDataRegPar_x[1].Description		:= ADR('Feeder Velocity');

	(* Filter files for pdf type *)
	MpFileManagerUIConnect.File.Filter	:= '*.pdf';
END_PROGRAM

PROGRAM _CYCLIC
	//***************************************************
	FOR i := 0 TO 49 DO
		// Save Filenames to a seperate array for display in Table
		DisplayFileName[i]											:= MpFileManagerUIConnect.File.List.Items[i].Name;
		// mark file selection
		MpFileManagerUIConnect.File.List.Items[i].IsSelected		:= (DisplayFileNameIndex = INT_TO_USINT(i));
	END_FOR
	StrSelectedFile := CONCAT(STR_FILE_DEVICE, MpFileManagerUIConnect.File.List.Items[DisplayFileNameIndex].Name);		// String for pdfViewer to display right report

	(* Configure visible file list *)
	brsstrcpy(ADR(TableConfig), ADR('{ "specRows": [{"from":'));
	brsitoa(MpFileManagerUIConnect.File.PathInfo.FileCount, ADR(TableConfig) + brsstrlen(ADR(TableConfig)));
	brsstrcat(ADR(TableConfig),  ADR(',"to":49, "visible":false}]}'));

	(* Call function blocks *)
	MpDataRecorder_0();
	FOR i := 0 TO MAX_IDX_DATA_REG DO
		MpDataRegPar_x[i]();
	END_FOR
	MpFileManagerUI_0();

	(* Reset ErrorReset command *)
	IF NOT MpDataRecorder_0.Error THEN
		MpDataRecorder_0.ErrorReset			:= FALSE;
	END_IF
	FOR i := 0 TO MAX_IDX_DATA_REG DO
		IF NOT MpDataRegPar_x[i].Error THEN
			MpDataRegPar_x[i].ErrorReset	:= FALSE;
		END_IF
	END_FOR
END_PROGRAM

PROGRAM _EXIT
	(* call mapp function blocks with enable = false *)
	MpFileManagerUI_0.Enable		:= FALSE;
	MpFileManagerUI_0();
	MpDataRecorder_0.Enable			:= FALSE;
	MpDataRecorder_0();
	FOR i := 0 TO MAX_IDX_DATA_REG DO
		MpDataRegPar_x[i].Enable	:= FALSE;
		MpDataRegPar_x[i]();
	END_FOR
END_PROGRAM
```

### Package Logical/Infrastructure/File - Package for mapp File Framework

### Program Logical/Infrastructure/File/FileMgr (IEC) - File manager

#### FileMgr.st - Init, cyclic, exit code
```iecst
//***********************************************************************
// Copyright: B&R Industrial Automation GmbH
// Author: B&R Industrial Automation GmbH
// Created: April 12, 2022
// Description: Task for file management
//***********************************************************************

PROGRAM _INIT

	// Inititialize mapp function block
	MpFileManagerUIConnect.DeviceList.DeviceNames[0] := 'mappRecipeFiles';
	MpFileManagerUIConnect.DeviceList.DeviceNames[1] := 'mappAuditFiles';
	MpFileManagerUIConnect.DeviceList.DeviceNames[2] := 'mappReportFiles';
	MpFileManagerUIConnect.DeviceList.DeviceNames[3] := 'mappDataFiles';
	MpFileManagerUIConnect.DeviceList.DeviceNames[4] := 'mappBackupFiles';
	MpFileManagerUIConnect.DeviceList.DeviceNames[5] := 'mappAlarmXFiles';
	MpFileManagerUIConnect.DeviceList.DeviceNames[6] := 'mappUserXFiles';
	MpFileManagerUI_0.Enable := TRUE;
	MpFileManagerUI_0.MpLink := ADR(gMpLinkFileManagerUIFile);
	MpFileManagerUI_0.UIConnect := ADR(MpFileManagerUIConnect);
	MpFileManagerUI_0.UISetup.FileListSize := SIZEOF(MpFileManagerUIConnect.File.List.Items) / SIZEOF(MpFileManagerUIConnect.File.List.Items[0]);
	MpFileManagerUI_0();

	// Initialize FIFO feature
    HmiFile.Parameters.Fifo.DeviceName := 'mappDataFiles';
    // MaxFolderSize is in kB
	HmiFile.Parameters.Fifo.MaxFolderSize := 20000;
    HmiFile.Parameters.Fifo.MaxNumberOfFiles := 20;
    // ScanInterval is in minutes
	HmiFile.Parameters.Fifo.ScanInterval := 60;

	// Initialize which folders should exist
	PathCheck.DeviceList := MpFileManagerUIConnect.DeviceList;
	PathCheck.Folder[0] := 'Recipe';
	PathCheck.Folder[1] := 'Audit';
	PathCheck.Folder[2] := 'Report';
	PathCheck.Folder[3] := 'Data';
	PathCheck.Folder[4] := 'Backup';
	PathCheck.Folder[5] := 'AlarmX';
	PathCheck.Folder[6] := 'UserX';

	HmiFile.Status.DeviceDataProvider[0] := '{"value":"mappRecipeFiles","text":"mappRecipeFiles"}';
	HmiFile.Status.DeviceDataProvider[1] := '{"value":"mappAuditFiles","text":"mappAuditFiles"}';
	HmiFile.Status.DeviceDataProvider[2] := '{"value":"mappReportFiles","text":"mappReportFiles"}';
	HmiFile.Status.DeviceDataProvider[3] := '{"value":"mappDataFiles","text":"mappDataFiles"}';
	HmiFile.Status.DeviceDataProvider[4] := '{"value":"mappBackupFiles","text":"mappBackupFiles"}';
	HmiFile.Status.DeviceDataProvider[5] := '{"value":"mappAlarmXFiles","text":"mappAlarmXFiles"}';
	HmiFile.Status.DeviceDataProvider[6] := '{"value":"mappUserXFiles","text":"mappUserXFiles"}';

	// Calculate offset for potential additional USB devices
	FOR i := 0 TO 9 DO
		IF MpFileManagerUIConnect.DeviceList.DeviceNames[i] <> '' THEN
			USBOffset := USBOffset + 1;
		END_IF
	END_FOR

END_PROGRAM

PROGRAM _CYCLIC

	// Call all actions
	FormatDeviceDataProvider;
	FileManager;
	IF HmiFile.Parameters.Fifo.Enable THEN
		FIFOOperation;
	END_IF

	// Error reset
    IF NOT MpFileManagerUI_0.Error THEN
        MpFileManagerUI_0.ErrorReset := FALSE;
    END_IF

	// Assign MpLink
	MpFileManagerUI_0.MpLink := ADR(gMpLinkFileManagerUIFile);

	// Call function block
	MpFileManagerUI_0();

END_PROGRAM

PROGRAM _EXIT

	// Disable the function blocls to unlink the MpLink
	MpFileManagerUI_0.Enable := FALSE;

	// Call function block
	MpFileManagerUI_0();

END_PROGRAM
```

#### FileMgr.typ - Local data types
```iecst
(*Structure types*)

TYPE
	FileHmiInterfaceType : 	STRUCT  (*Structure to hold commands, parameters and status from the HMI*)
		Commands : FileHmiCommandsType; (*Structure to hold the commands from the HMI*)
		Parameters : FileHmiParametersType; (*Structure to hold parameters for the mapp View HMI*)
		Status : FileHmiStatusType; (*Structure to hold status information from the mapp View HMI*)
	END_STRUCT;
	FileHmiCommandsType : 	STRUCT  (*Structure to hold the commands from the HMI*)
		Delete : BOOL; (*Delete file*)
		FolderUp : BOOL; (*Move back/up a folder*)
		EnterFolder : BOOL; (*Move forward/down a folder*)
		MultiSelect : BOOL; (*Enables the ability to select multiple files*)
		CheckFolder : BOOL; (*Run the FIFO check to determine if old files should be deleted*)
	END_STRUCT;
	FileHmiParametersType : 	STRUCT  (*Structure to hold parameters for the mapp View HMI*)
		OldSortOrder : MpFileManagerUISortOrderEnum; (*Previous sord order*)
		Fifo : FileHmiParaFifoType; (*Parameters for the FIFO feature (first-in-first-out)*)
	END_STRUCT;
	FileHmiStatusType : 	STRUCT  (*Structure to hold status information from the mapp View HMI*)
		FileNames : ARRAY[0..49]OF STRING[80]; (*List of file names*)
		TimeStamps : ARRAY[0..49]OF DATE_AND_TIME; (*List of time stamps for file names*)
		Type : ARRAY[0..49]OF DINT; (*List of file types*)
		Size : ARRAY[0..49]OF UDINT; (*List of file sizes*)
		DeviceDataProvider : ARRAY[0..MAX_IDX_FILE_DEV]OF STRING[100]; (*Data provider for the file device selector*)
		DeviceName : STRING[50]; (*File device name*)
		FileName : STRING[255]; (*Fille name*)
		TableConfig : ARRAY[0..1]OF STRING[120]; (*Table configuration for the file explorer (table widget) on the mapp View HMI*)
		IsFolder : BOOL; (*Flag for whether the item is a folder (versus a file)*)
		BackButton : BOOL; (*Flag for whether the back button should be shown*)
		DeleteStep : FileDeleteStepEnum; (*Enumeration for automatic file deletion steps*)
		AutoDeleteSelected : USINT; (*Number of selected items*)
		FolderSize : REAL; (*Size of currently selected folder*)
		SelectedIndex : USINT; (*Selected index in the file list*)
		CurrentPage : STRING[80]; (*Current page*)
	END_STRUCT;
	FileHmiParaFifoType : 	STRUCT  (*Parameters for the FIFO feature (first-in-first-out)*)
		Enable : BOOL; (*FIFO enable*)
		DeviceName : STRING[50]; (*File device that the FIFO is active on*)
		FifoType : FileFifoTypeEnum; (*Defines the delete behavior of the FIFO*)
		ScanInterval : DINT := 60; (*[minutes]*)
		MaxFileAge : UINT := 365; (*[days] Files older than 1 year will be deleted*)
		MaxFolderSize : REAL := 1000; (*[kB] - Max size of files inside the active folder*)
		MaxNumberOfFiles : UINT := 20; (*Max number of files inside active folder*)
	END_STRUCT;
END_TYPE

(*Enumerations*)

TYPE
	FileDeleteStepEnum :
		( (*Enumeration for file deletion steps*)
		FILE_DELETE_WAIT := 0, (*Wait state*)
		FILE_SCAN_FOLDER_WAIT, (*Wait for check for old files command*)
		FILE_SELECT_DEVICE, (*Switch file device to the configured one *)
		FILE_SORT_BY_DATE, (*Sort by date so the oldest files are at the end*)
		FILE_SORT_BY_DATE_WAIT, (*Wait step switching sorting mode*)
		FILE_CHECK_FOR_FILTER, (*Check which delete filter is active*)
		FILE_SELECT_OLDEST_FILES_0, (*Scan and select all file over the filter setting*)
		FILE_CALC_FOLDER_SIZE, (*Calculate the overall file size in the open folder*)
		FILE_SELECT_OLDEST_FILES_1, (*Scan and select all file over the filter setting*)
		FILE_DELETE_FILES, (*Set command to delete the selected oldest files*)
		FILE_CONFIRM_DELETE, (*Confirm the file delete*)
		FILE_RESET_SORT_BY, (*Restore old sort order*)
		FILE_RESET_SORT_BY_WAIT (*Waiting for restore previous sort order*)
		);
	FileFifoTypeEnum :
		( (*Defines the delete behavior of the FIFO*)
		FILE_FIFO_NUM_OF_FILES := 0, (*Delete according to total number of files*)
		FILE_FIFO_SIZE_OF_FOLDER (*Delete according to maximum folder size*)
		);
	FileTypeEnum :
		( (*Defines the type of file in order to update the displayed icon*)
		FOLDER := 0, (*Folder*)
		FILE := 1, (*File*)
		FILE_SELECTED := 2 (*The selected file*)
		);
END_TYPE
```

#### FileMgr.var - Local variables
```iecst
(*Function Blocks*)
VAR
	MpFileManagerUI_0 : MpFileManagerUI; (*MpFileManagerUI instance*)
	DirInfo_0 : DirInfo;
	R_TRIG_CheckStatus : R_TRIG;
	TON_ScanFolder : TON;
END_VAR
(*Constants*)
VAR CONSTANT
	MAX_IDX_FILE_DEV : USINT := MAX_IDX_USB_DEV_LIST + 7; (*Maximum number of  file devices *)
END_VAR
(*Structure Types*)
VAR
	MpFileManagerUIConnect : MpFileManagerUIConnectType; (*File manager connection to the HMI*)
	HmiFile : FileHmiInterfaceType; (*HMI interface structure*)
END_VAR
(*Variables*)
VAR
	i : USINT; (*Index for FOR loops*)
	DeviceListCount : USINT; (*Counter for accessible file devices*)
	DeviceCount : USINT; (*Counter for available file devices*)
	Index : USINT; (*Index for avaliable devices*)
	FolderDepthCount : USINT; (*Keeps track of the folder depth location to determine whether or not the back button should be shown*)
	PathCheck : FilePathCheckType;
	USBOffset : USINT := 0; (*Device list offset where to add USB device*)
END_VAR
```

#### HMIActions.st
```iecst
ACTION FormatDeviceDataProvider:

	// Select CF device if USB device is not available
    FOR i := 0 TO MAX_IDX_USB_DEV_LIST DO
        IF gUSBAvailable[i] THEN

			HmiFile.Status.DeviceDataProvider[i + 7] := '{"value":"USB';
            brsitoa(i + 1, ADR(HmiFile.Status.DeviceDataProvider[i + 7]) + brsstrlen(ADR(HmiFile.Status.DeviceDataProvider[i + 7])));

			brsstrcat(ADR(HmiFile.Status.DeviceDataProvider[i + 7]), ADR('","text":"USB'));
            brsitoa(i + 1, ADR(HmiFile.Status.DeviceDataProvider[i + 7]) + brsstrlen(ADR(HmiFile.Status.DeviceDataProvider[i + 7])));
            brsstrcat(ADR(HmiFile.Status.DeviceDataProvider[i + 7]), ADR('"}'));

			MpFileManagerUIConnect.DeviceList.DeviceNames[i + 7] := 'USB';
            brsitoa(i + 1, ADR(MpFileManagerUIConnect.DeviceList.DeviceNames[i + 7]) + brsstrlen(ADR(MpFileManagerUIConnect.DeviceList.DeviceNames[i + 7])));
        ELSE
            brsmemset(ADR(HmiFile.Status.DeviceDataProvider[i + 7]), 0, SIZEOF(HmiFile.Status.DeviceDataProvider[i + 7]));
            brsmemset(ADR(MpFileManagerUIConnect.DeviceList.DeviceNames[i + 7]), 0, SIZEOF(MpFileManagerUIConnect.DeviceList.DeviceNames[i + 7]));
        END_IF
    END_FOR

	//Check initilized folder for existance and remove any from the device list that don't exist
	IF DirInfo_0.status = ERR_OK  THEN
		IF PathCheck.DeviceList.DeviceNames[DeviceListCount] = '' THEN
			//Delete entries past the actual number of devices found
			FOR i:=Index TO 9 DO
				MpFileManagerUIConnect.DeviceList.DeviceNames[i] := '';
			END_FOR
			Index := 0;
			DeviceListCount := 0;
		END_IF
		// copy device name from source list into the actual device list
		MpFileManagerUIConnect.DeviceList.DeviceNames[Index] := PathCheck.DeviceList.DeviceNames[DeviceListCount];
		Index := Index + 1;

		DeviceListCount := DeviceListCount + 1;
		IF DeviceListCount > 9 THEN
			DeviceListCount := 0;
		END_IF
		IF Index > 9 THEN
			Index := 0;
		END_IF
	ELSIF DirInfo_0.status = fiERR_DIR_NOT_EXIST  THEN
		DeviceListCount := DeviceListCount + 1;
		IF DeviceListCount > 9 THEN
			DeviceListCount := 0;
		END_IF
	END_IF

	DirInfo_0(enable:= TRUE, pDevice := ADR('UserPartition'), pPath := ADR(PathCheck.Folder[DeviceListCount]));

	// Configure visible device list
	HmiFile.Status.TableConfig[0] := '{ "specRows": [{"from":';
	FOR i := 0 TO 9 DO
		IF MpFileManagerUIConnect.DeviceList.DeviceNames[i] <> '' THEN
			DeviceCount := i + 1;
		END_IF
	END_FOR
	brsitoa((DeviceCount), ADR(HmiFile.Status.TableConfig[0]) + brsstrlen(ADR(HmiFile.Status.TableConfig[0])));
    brsstrcat(ADR(HmiFile.Status.TableConfig[0]),  ADR(',"to":9, "visible":false}]}'));

    // Configure visible file list
	HmiFile.Status.TableConfig[1] := '{ "specRows": [{"from":';
    brsitoa((MpFileManagerUIConnect.File.PathInfo.FileCount + MpFileManagerUIConnect.File.PathInfo.FolderCount), ADR(HmiFile.Status.TableConfig[1]) + brsstrlen(ADR(HmiFile.Status.TableConfig[1])));
    brsstrcat(ADR(HmiFile.Status.TableConfig[1]),  ADR(',"to":49, "visible":false}]}'));

END_ACTION

ACTION FileManager:

    MpFileManagerUI_0.MpLink := ADR(gMpLinkFileManagerUIFile);
    MpFileManagerUI_0.UIConnect := ADR(MpFileManagerUIConnect);
	MpFileManagerUI_0();

    FOR i := 0 TO ((SIZEOF(HmiFile.Status.FileNames)/SIZEOF(HmiFile.Status.FileNames[0])) - 1) DO
        HmiFile.Status.FileNames[i] := MpFileManagerUIConnect.File.List.Items[i].Name;
        HmiFile.Status.TimeStamps[i] := MpFileManagerUIConnect.File.List.Items[i].LastModified;
        HmiFile.Status.Size[i] := REAL_TO_UDINT(UDINT_TO_REAL(MpFileManagerUIConnect.File.List.Items[i].Size) * 0.001);

		// Set image array based on item type
		IF MpFileManagerUIConnect.File.List.Items[i].IsFolder THEN
			HmiFile.Status.Type[i] := FOLDER;
		ELSIF NOT MpFileManagerUIConnect.File.List.Items[i].IsFolder AND MpFileManagerUIConnect.File.List.Items[i].IsSelected THEN
			HmiFile.Status.Type[i] := FILE_SELECTED;
		ELSE
			HmiFile.Status.Type[i] := FILE;
		END_IF

		// Set file selected when the table is clicked Single and MultiSelect
		IF HmiFile.Status.DeleteStep = FILE_DELETE_WAIT THEN
			IF (MpFileManagerUIConnect.File.MultiSelect = FALSE) THEN
				IF (i = HmiFile.Status.SelectedIndex) THEN
					MpFileManagerUIConnect.File.List.Items[i].IsSelected := TRUE;
				ELSE
					MpFileManagerUIConnect.File.List.Items[i].IsSelected := FALSE;
				END_IF
			ELSIF (MpFileManagerUIConnect.File.MultiSelect = TRUE) AND HmiFile.Commands.MultiSelect THEN
				IF (i = HmiFile.Status.SelectedIndex) AND NOT MpFileManagerUIConnect.File.List.Items[i].IsSelected THEN
					MpFileManagerUIConnect.File.List.Items[i].IsSelected := TRUE;
					HmiFile.Commands.MultiSelect := FALSE;
				ELSIF (i = HmiFile.Status.SelectedIndex) AND MpFileManagerUIConnect.File.List.Items[i].IsSelected THEN
					MpFileManagerUIConnect.File.List.Items[i].IsSelected := FALSE;
					HmiFile.Commands.MultiSelect := FALSE;
				END_IF
			END_IF
		END_IF
    END_FOR

	// Read currently selected device name for HMI
	HmiFile.Status.DeviceName := MpFileManagerUIConnect.DeviceList.DeviceNames[MpFileManagerUIConnect.DeviceList.SelectedIndex];

	// Read if current selected object is folder
	HmiFile.Status.IsFolder := MpFileManagerUIConnect.File.List.Items[HmiFile.Status.SelectedIndex].IsFolder;

	// Control the folder structure when entering and leaving folders
	IF (HmiFile.Commands.EnterFolder) AND MpFileManagerUIConnect.File.List.Items[HmiFile.Status.SelectedIndex].IsFolder THEN
		HmiFile.Commands.EnterFolder := FALSE;
		MpFileManagerUIConnect.File.EnterFolder := TRUE;
		FolderDepthCount := FolderDepthCount + 1;
	ELSE
		HmiFile.Commands.EnterFolder := FALSE;
	END_IF

	IF EDGEPOS(HmiFile.Commands.FolderUp) AND (HmiFile.Status.BackButton > 0) THEN
		HmiFile.Commands.FolderUp := FALSE;
		MpFileManagerUIConnect.File.FolderUp := TRUE;
		FolderDepthCount := FolderDepthCount - 1;
	END_IF

	IF FolderDepthCount > 0 THEN
		HmiFile.Status.BackButton := TRUE;
	ELSE
		HmiFile.Status.BackButton := FALSE;
	END_IF

END_ACTION
```

#### FIFOOperations.st
```iecst
ACTION FIFOOperation:

	R_TRIG_CheckStatus(CLK := (MpFileManagerUIConnect.Status = mpFILE_UI_STATUS_CHANGE_DIR) OR
		(MpFileManagerUIConnect.Status = mpFILE_UI_STATUS_CHANGE_DEVICE) OR
		(MpFileManagerUIConnect.Status = mpFILE_UI_STATUS_CREATE));

	IF R_TRIG_CheckStatus.Q OR TON_ScanFolder.Q THEN
		HmiFile.Commands.CheckFolder := TRUE;
	END_IF

	// Autodelete oldest files based on scanning option
    CASE HmiFile.Status.DeleteStep OF

		FILE_DELETE_WAIT:
			// Wait for check the correct device selection
			TON_ScanFolder.IN := (HmiFile.Status.CurrentPage <> 'File_page');
			IF TON_ScanFolder.Q THEN
				TON_ScanFolder.IN := FALSE;
				HmiFile.Status.DeleteStep := FILE_SCAN_FOLDER_WAIT;
			END_IF

		FILE_SCAN_FOLDER_WAIT:
			// Wait for check for old files command
			IF (HmiFile.Commands.CheckFolder = TRUE) AND (MpFileManagerUIConnect.Status = mpFILE_UI_STATUS_IDLE) THEN
				HmiFile.Commands.CheckFolder := FALSE;
				HmiFile.Status.DeleteStep := FILE_SELECT_DEVICE;
				HmiFile.Parameters.OldSortOrder := MpFileManagerUIConnect.File.SortOrder;
			END_IF

		FILE_SELECT_DEVICE:
			//
            IF (HmiFile.Status.DeviceName <> HmiFile.Parameters.Fifo.DeviceName) THEN
				FOR i := 0 TO ((SIZEOF(MpFileManagerUIConnect.DeviceList.DeviceNames)/SIZEOF(MpFileManagerUIConnect.DeviceList.DeviceNames[0])) - 1) DO
        			IF HmiFile.Parameters.Fifo.DeviceName = MpFileManagerUIConnect.DeviceList.DeviceNames[i] THEN
						MpFileManagerUIConnect.DeviceList.SelectedIndex := i;
					END_IF
    			END_FOR
            END_IF

            IF (HmiFile.Status.DeviceName = HmiFile.Parameters.Fifo.DeviceName) AND (MpFileManagerUIConnect.Status = mpFILE_UI_STATUS_IDLE) THEN
                HmiFile.Status.DeleteStep := FILE_SORT_BY_DATE;
            END_IF

		FILE_SORT_BY_DATE:
			// Sort by date so the oldest files are at the end
            IF (MpFileManagerUIConnect.File.SortOrder <> mpFILE_SORT_BY_MOD_TIME_DESC) THEN
                MpFileManagerUIConnect.File.SortOrder := mpFILE_SORT_BY_MOD_TIME_DESC;
            ELSIF (MpFileManagerUIConnect.Status = mpFILE_UI_STATUS_IDLE) THEN
                MpFileManagerUIConnect.File.Refresh := TRUE;
            END_IF

			IF (MpFileManagerUIConnect.Status = mpFILE_UI_STATUS_REFRESH) AND (MpFileManagerUIConnect.File.Refresh = FALSE) THEN
                HmiFile.Status.DeleteStep := FILE_SORT_BY_DATE_WAIT;
            END_IF

       FILE_SORT_BY_DATE_WAIT:
	        // Wait for the file manager to complete sorting change
            IF (MpFileManagerUIConnect.Status = mpFILE_UI_STATUS_IDLE) THEN
                HmiFile.Status.DeleteStep := FILE_CHECK_FOR_FILTER;
            END_IF

		FILE_CHECK_FOR_FILTER:
			// Check which delete filter is active
            IF (HmiFile.Parameters.Fifo.FifoType = FILE_FIFO_NUM_OF_FILES) THEN
                HmiFile.Status.DeleteStep := FILE_SELECT_OLDEST_FILES_0;
            ELSIF (HmiFile.Parameters.Fifo.FifoType = FILE_FIFO_SIZE_OF_FOLDER) THEN
				HmiFile.Status.DeleteStep := FILE_CALC_FOLDER_SIZE;
            END_IF

        FILE_SELECT_OLDEST_FILES_0:
			// Scan and select all file over the filter setting
			IF (MpFileManagerUIConnect.Status = mpFILE_UI_STATUS_IDLE) THEN
				IF MpFileManagerUIConnect.File.PathInfo.FileCount > 1 THEN
           			MpFileManagerUIConnect.File.MultiSelect := TRUE;
				END_IF
				HmiFile.Status.AutoDeleteSelected := 0;
				FOR i := 0 TO ((SIZEOF(HmiFile.Status.FileNames)/SIZEOF(HmiFile.Status.FileNames[0])) - 1) DO
					IF i >= HmiFile.Parameters.Fifo.MaxNumberOfFiles THEN
						MpFileManagerUIConnect.File.List.Items[0].IsSelected := FALSE;
						IF (MpFileManagerUIConnect.File.List.Items[i].ItemType <> mpFILE_ITEM_TYPE_NONE) AND NOT MpFileManagerUIConnect.File.List.Items[i].IsFolder THEN
							MpFileManagerUIConnect.File.List.Items[i].IsSelected := TRUE;
							HmiFile.Status.AutoDeleteSelected := HmiFile.Status.AutoDeleteSelected + 1;
						END_IF
					END_IF
				END_FOR

				IF (HmiFile.Status.AutoDeleteSelected > 0) THEN
					HmiFile.Status.DeleteStep := FILE_DELETE_FILES;
				ELSE
					MpFileManagerUIConnect.File.MultiSelect := FALSE;
					HmiFile.Status.DeleteStep := FILE_RESET_SORT_BY;
				END_IF
			END_IF

		FILE_CALC_FOLDER_SIZE:
			// Calculate the overall file size in the open folder
				HmiFile.Status.FolderSize := 0;
				FOR i := 0 TO ((SIZEOF(HmiFile.Status.FileNames)/SIZEOF(HmiFile.Status.FileNames[0])) - 1) DO
					IF MpFileManagerUIConnect.File.List.Items[i].ItemType <> mpFILE_ITEM_TYPE_FOLDER THEN
						HmiFile.Status.FolderSize := HmiFile.Status.FolderSize + UDINT_TO_REAL(MpFileManagerUIConnect.File.List.Items[i].Size);
					END_IF
				END_FOR
				IF (HmiFile.Status.FolderSize > HmiFile.Parameters.Fifo.MaxFolderSize) THEN
					HmiFile.Status.DeleteStep := FILE_SELECT_OLDEST_FILES_1;
				ELSE
					HmiFile.Status.DeleteStep := FILE_RESET_SORT_BY;
				END_IF

		FILE_SELECT_OLDEST_FILES_1:
			// Scan and select all file over the filter setting
			IF (MpFileManagerUIConnect.Status = mpFILE_UI_STATUS_IDLE) THEN
				MpFileManagerUIConnect.File.List.Items[(MpFileManagerUIConnect.File.PathInfo.FileCount - 1)].IsSelected := TRUE;
				HmiFile.Status.DeleteStep := FILE_DELETE_FILES;
			END_IF

		FILE_DELETE_FILES:
			// Set command to delete the selected oldest files
			IF  (MpFileManagerUIConnect.Status = mpFILE_UI_STATUS_IDLE) THEN
				MpFileManagerUIConnect.File.Delete := TRUE;
			END_IF

			IF (MpFileManagerUIConnect.Status = mpFILE_UI_STATUS_DELETE) THEN
				HmiFile.Status.DeleteStep := FILE_CONFIRM_DELETE;
            END_IF

		FILE_CONFIRM_DELETE:
			// Confirm the file delete
            IF (MpFileManagerUIConnect.MessageBox.Type = mpFILE_MSG_CONFIRM_DELETE) THEN
                MpFileManagerUIConnect.MessageBox.Confirm := TRUE;
            ELSIF (MpFileManagerUIConnect.Status = mpFILE_UI_STATUS_IDLE) AND (MpFileManagerUIConnect.MessageBox.LayerStatus = 1) THEN
				IF (HmiFile.Parameters.Fifo.FifoType = FILE_FIFO_SIZE_OF_FOLDER) THEN
                	HmiFile.Status.DeleteStep := FILE_CALC_FOLDER_SIZE;
				ELSE
					HmiFile.Status.DeleteStep := FILE_RESET_SORT_BY;
					MpFileManagerUIConnect.File.MultiSelect := FALSE;
				END_IF
            END_IF

		FILE_RESET_SORT_BY:
			// Restore old sort order
            IF (MpFileManagerUIConnect.File.SortOrder <> HmiFile.Parameters.OldSortOrder) THEN
                MpFileManagerUIConnect.File.SortOrder := HmiFile.Parameters.OldSortOrder;
            ELSIF (MpFileManagerUIConnect.Status = mpFILE_UI_STATUS_IDLE) THEN
                MpFileManagerUIConnect.File.Refresh := TRUE;
				HmiFile.Status.DeleteStep := FILE_RESET_SORT_BY_WAIT;
            END_IF

		FILE_RESET_SORT_BY_WAIT:
			// Wait for file manager to complete restoring previous sorting mode
            IF (MpFileManagerUIConnect.Status = mpFILE_UI_STATUS_REFRESH) OR (MpFileManagerUIConnect.Status = mpFILE_UI_STATUS_IDLE) THEN
                HmiFile.Status.DeleteStep := FILE_DELETE_WAIT;
				IF (MpFileManagerUIConnect.MessageBox.Type = mpFILE_MSG_BUSY) THEN
					MpFileManagerUIConnect.MessageBox.Confirm := TRUE;
				END_IF
            END_IF
	END_CASE

	// Timer to scan file device in intervals
	TON_ScanFolder(PT := DINT_TO_TIME(HmiFile.Parameters.Fifo.ScanInterval * 60000));

END_ACTION
```

### Program Logical/Infrastructure/File/File (IEC)

#### FileMgt.st - Init, cyclic, exit code
```iecst
//***********************************************************************
// Copyright: B&R Industrial Automation GmbH
// Author: B&R Industrial Automation GmbH
// Created: Jan 1, 2022
// Description: Tasks for File management control. The File management
// handling is done in this task.
//***********************************************************************

PROGRAM _INIT

	// Inititialize mapp function block
	MpFileManagerUIConnect.DeviceList.DeviceNames[0] := 'mappRecipeFiles';
	MpFileManagerUIConnect.DeviceList.DeviceNames[1] := 'mappAuditFiles';
	MpFileManagerUIConnect.DeviceList.DeviceNames[2] := 'mappReportFiles';
	MpFileManagerUIConnect.DeviceList.DeviceNames[3] := 'mappDataFiles';
	MpFileManagerUIConnect.DeviceList.DeviceNames[4] := 'mappBackupFiles';
	MpFileManagerUIConnect.DeviceList.DeviceNames[5] := 'mappAlarmXFiles';
	MpFileManagerUIConnect.DeviceList.DeviceNames[6] := 'mappUserXFiles';
	MpFileManagerUI_0.Enable := TRUE;
	MpFileManagerUI_0.MpLink := ADR(gMpLinkFileManagerUIFile);
	MpFileManagerUI_0.UIConnect := ADR(MpFileManagerUIConnect);
	MpFileManagerUI_0.UISetup.FileListSize := SIZEOF(MpFileManagerUIConnect.File.List.Items) / SIZEOF(MpFileManagerUIConnect.File.List.Items[0]);
	MpFileManagerUI_0();

	// Initialize FIFO feature
    HmiFile.Parameters.Fifo.DeviceName := 'mappDataFiles';
    // MaxFolderSize is in kB
	HmiFile.Parameters.Fifo.MaxFolderSize := 20000;
    HmiFile.Parameters.Fifo.MaxNumberOfFiles := 20;
    // ScanInterval is in minutes
	HmiFile.Parameters.Fifo.ScanInterval := 60;

	HmiFile.Status.DeviceDataProvider[0] := '{"value":"mappRecipe","text":"mappRecipe"}';
	HmiFile.Status.DeviceDataProvider[1] := '{"value":"mappAudit","text":"mappAudit"}';
	HmiFile.Status.DeviceDataProvider[2] := '{"value":"mappReport","text":"mappReport"}';
	HmiFile.Status.DeviceDataProvider[3] := '{"value":"mappData","text":"mappData"}';
	HmiFile.Status.DeviceDataProvider[4] := '{"value":"mappBackup","text":"mappBackup"}';
	HmiFile.Status.DeviceDataProvider[5] := '{"value":"mappAlarmX","text":"mappAlarmX"}';
	HmiFile.Status.DeviceDataProvider[6] := '{"value":"mappUserX","text":"mappUserX"}';

END_PROGRAM

PROGRAM _CYCLIC

	// Call all actions
	FormatDeviceDataProvider;
	FileManager;
	IF HmiFile.Parameters.Fifo.Enable THEN
		FIFOOperation;
	END_IF

	// Error reset
    IF NOT MpFileManagerUI_0.Error THEN
        MpFileManagerUI_0.ErrorReset := FALSE;
    END_IF

	// Assign MpLink
	MpFileManagerUI_0.MpLink := ADR(gMpLinkFileManagerUIFile);

	// Call function block
	MpFileManagerUI_0();

END_PROGRAM

PROGRAM _EXIT

	// Disable the function blocls to unlink the MpLink
	MpFileManagerUI_0.Enable := FALSE;

	// Call function block
	MpFileManagerUI_0();

END_PROGRAM
```

#### HMIActions.st
```iecst
ACTION FormatDeviceDataProvider:

	// Select CF device if USB device is not available
    FOR Index := 0 TO MAX_IDX_USB_DEV_LIST DO
        IF gUSBAvailable[Index] THEN

            brsstrcpy(ADR(HmiFile.Status.DeviceDataProvider[Index + 7]), ADR('{"value":"USB'));
            brsitoa(Index + 1, ADR(HmiFile.Status.DeviceDataProvider[Index + 7]) + brsstrlen(ADR(HmiFile.Status.DeviceDataProvider[Index + 7])));

			brsstrcat(ADR(HmiFile.Status.DeviceDataProvider[Index + 7]), ADR('","text":"USB'));
            brsitoa(Index + 1, ADR(HmiFile.Status.DeviceDataProvider[Index + 7]) + brsstrlen(ADR(HmiFile.Status.DeviceDataProvider[Index + 7])));
            brsstrcat(ADR(HmiFile.Status.DeviceDataProvider[Index + 7]), ADR('"}'));

		    brsstrcpy(ADR(MpFileManagerUIConnect.DeviceList.DeviceNames[Index + 7]), ADR('USB'));
            brsitoa(Index + 1, ADR(MpFileManagerUIConnect.DeviceList.DeviceNames[Index + 7]) + brsstrlen(ADR(MpFileManagerUIConnect.DeviceList.DeviceNames[Index + 7])));
        ELSE
            brsmemset(ADR(HmiFile.Status.DeviceDataProvider[Index + 7]), 0, SIZEOF(HmiFile.Status.DeviceDataProvider[Index + 7]));
            brsmemset(ADR(MpFileManagerUIConnect.DeviceList.DeviceNames[Index + 7]), 0, SIZEOF(MpFileManagerUIConnect.DeviceList.DeviceNames[Index + 7]));
        END_IF
    END_FOR

	// Configure visible device list
    brsstrcpy(ADR(HmiFile.Status.TableConfig[0]), ADR('{ "specRows": [{"from":'));
	FOR i := 0 TO 9 DO
		IF MpFileManagerUIConnect.DeviceList.DeviceNames[i] <> '' THEN
			DeviceCount := i + 1;
		END_IF
	END_FOR
	brsitoa((DeviceCount), ADR(HmiFile.Status.TableConfig[0]) + brsstrlen(ADR(HmiFile.Status.TableConfig[0])));
    brsstrcat(ADR(HmiFile.Status.TableConfig[0]),  ADR(',"to":9, "visible":false}]}'));

    // Configure visible file list
    brsstrcpy(ADR(HmiFile.Status.TableConfig[1]), ADR('{ "specRows": [{"from":'));
    brsitoa((MpFileManagerUIConnect.File.PathInfo.FileCount + MpFileManagerUIConnect.File.PathInfo.FolderCount), ADR(HmiFile.Status.TableConfig[1]) + brsstrlen(ADR(HmiFile.Status.TableConfig[1])));
    brsstrcat(ADR(HmiFile.Status.TableConfig[1]),  ADR(',"to":49, "visible":false}]}'));

END_ACTION

ACTION FileManager:

    MpFileManagerUI_0.MpLink := ADR(gMpLinkFileManagerUIFile);
    MpFileManagerUI_0.UIConnect := ADR(MpFileManagerUIConnect);
    MpFileManagerUI_0();
    FOR i := 0 TO ((SIZEOF(HmiFile.Status.FileNames)/SIZEOF(HmiFile.Status.FileNames[0])) - 1) DO
        HmiFile.Status.FileNames[i] := MpFileManagerUIConnect.File.List.Items[i].Name;
        HmiFile.Status.TimeStamps[i] := MpFileManagerUIConnect.File.List.Items[i].LastModified;
        HmiFile.Status.Size[i] := REAL_TO_UDINT(UDINT_TO_REAL(MpFileManagerUIConnect.File.List.Items[i].Size) * 0.001);

		// Set image array based on item type
		IF MpFileManagerUIConnect.File.List.Items[i].IsFolder THEN
			HmiFile.Status.Type[i] := FOLDER;
		ELSIF NOT MpFileManagerUIConnect.File.List.Items[i].IsFolder AND MpFileManagerUIConnect.File.List.Items[i].IsSelected THEN
			HmiFile.Status.Type[i] := FILE_SELECTED;
		ELSE
			HmiFile.Status.Type[i] := FILE;
		END_IF

		// Set file selected when the table is clicked Single and MultiSelect
		IF HmiFile.Status.DeleteStep = FILE_DELETE_WAIT THEN
			IF (MpFileManagerUIConnect.File.MultiSelect = FALSE) THEN
				IF (i = HmiFile.Parameters.SelectedIndex) THEN
					MpFileManagerUIConnect.File.List.Items[i].IsSelected := TRUE;
				ELSE
					MpFileManagerUIConnect.File.List.Items[i].IsSelected := FALSE;
				END_IF
			ELSIF (MpFileManagerUIConnect.File.MultiSelect = TRUE) AND HmiFile.Commands.MultiSelect THEN
				IF (i = HmiFile.Parameters.SelectedIndex) AND NOT MpFileManagerUIConnect.File.List.Items[i].IsSelected THEN
					MpFileManagerUIConnect.File.List.Items[i].IsSelected := TRUE;
					HmiFile.Commands.MultiSelect := FALSE;
				ELSIF (i = HmiFile.Parameters.SelectedIndex) AND MpFileManagerUIConnect.File.List.Items[i].IsSelected THEN
					MpFileManagerUIConnect.File.List.Items[i].IsSelected := FALSE;
					HmiFile.Commands.MultiSelect := FALSE;
				END_IF
			END_IF
		END_IF
    END_FOR

	// Read currently selected device name for HMI
	HmiFile.Status.DeviceName := MpFileManagerUIConnect.DeviceList.DeviceNames[MpFileManagerUIConnect.DeviceList.SelectedIndex];

	// Read if current selected object is folder
	HmiFile.Status.IsFolder := MpFileManagerUIConnect.File.List.Items[HmiFile.Parameters.SelectedIndex].IsFolder;

	// Control the folder structure when entering and leaving folders
	IF (HmiFile.Commands.EnterFolder) AND MpFileManagerUIConnect.File.List.Items[HmiFile.Parameters.SelectedIndex].IsFolder THEN
		HmiFile.Commands.EnterFolder := FALSE;
		MpFileManagerUIConnect.File.EnterFolder := TRUE;
		FolderDepthCount := FolderDepthCount + 1;
	ELSE
		HmiFile.Commands.EnterFolder := FALSE;
	END_IF

	IF EDGEPOS(HmiFile.Commands.FolderUp) AND (HmiFile.Status.BackButton > 0) THEN
		HmiFile.Commands.FolderUp := FALSE;
		MpFileManagerUIConnect.File.FolderUp := TRUE;
		FolderDepthCount := FolderDepthCount - 1;
	END_IF

	IF FolderDepthCount > 0 THEN
		HmiFile.Status.BackButton := TRUE;
	ELSE
		HmiFile.Status.BackButton := FALSE;
	END_IF

END_ACTION
```

#### FIFOOperations.st
```iecst
ACTION FIFOOperation:

	R_TRIG_CheckStatus(CLK := (MpFileManagerUIConnect.Status = mpFILE_UI_STATUS_CHANGE_DIR) OR
		(MpFileManagerUIConnect.Status = mpFILE_UI_STATUS_CHANGE_DEVICE) OR
		(MpFileManagerUIConnect.Status = mpFILE_UI_STATUS_CREATE));

	IF R_TRIG_CheckStatus.Q OR TON_ScanFolder.Q THEN
		HmiFile.Commands.CheckFolder := TRUE;
	END_IF

	// Autodelete oldest files based on scanning option
    CASE HmiFile.Status.DeleteStep OF

		FILE_DELETE_WAIT:
			// Wait for check the correct device selection
			TON_ScanFolder.IN := (HmiFile.Status.CurrentPage <> 'File_page');
			IF TON_ScanFolder.Q THEN
				TON_ScanFolder.IN := FALSE;
				HmiFile.Status.DeleteStep := FILE_SCAN_FOLDER_WAIT;
			END_IF

		FILE_SCAN_FOLDER_WAIT:
			// Wait for check for old files command
			IF (HmiFile.Commands.CheckFolder = TRUE) AND (MpFileManagerUIConnect.Status = mpFILE_UI_STATUS_IDLE) THEN
				HmiFile.Commands.CheckFolder := FALSE;
				HmiFile.Status.DeleteStep := FILE_SELECT_DEVICE;
				HmiFile.Parameters.OldSortOrder := MpFileManagerUIConnect.File.SortOrder;
			END_IF

		FILE_SELECT_DEVICE:
			// Sort by date so the oldest files are at the end
            IF (HmiFile.Status.DeviceName <> HmiFile.Parameters.Fifo.DeviceName) THEN
				FOR i := 0 TO ((SIZEOF(MpFileManagerUIConnect.DeviceList.DeviceNames)/SIZEOF(MpFileManagerUIConnect.DeviceList.DeviceNames[0])) - 1) DO
        			IF HmiFile.Parameters.Fifo.DeviceName = MpFileManagerUIConnect.DeviceList.DeviceNames[i] THEN
						MpFileManagerUIConnect.DeviceList.SelectedIndex := i;
					END_IF
    			END_FOR
            END_IF

            IF (HmiFile.Status.DeviceName = HmiFile.Parameters.Fifo.DeviceName) AND (MpFileManagerUIConnect.Status = mpFILE_UI_STATUS_IDLE) THEN
                HmiFile.Status.DeleteStep := FILE_SORT_BY_DATE;
            END_IF

		FILE_SORT_BY_DATE:
			// Sort by date so the oldest files are at the end
            IF (MpFileManagerUIConnect.File.SortOrder <> mpFILE_SORT_BY_MOD_TIME_DESC) THEN
                MpFileManagerUIConnect.File.SortOrder := mpFILE_SORT_BY_MOD_TIME_DESC;
            ELSIF (MpFileManagerUIConnect.Status = mpFILE_UI_STATUS_IDLE) THEN
                MpFileManagerUIConnect.File.Refresh := TRUE;
            END_IF

            IF (MpFileManagerUIConnect.Status = mpFILE_UI_STATUS_REFRESH) THEN
                HmiFile.Status.DeleteStep := FILE_CHECK_FOR_FILTER;
            END_IF

		FILE_CHECK_FOR_FILTER:
			// Check which delete filter is active
            IF (HmiFile.Parameters.Fifo.FifoType = FILE_FIFO_NUM_OF_FILES) THEN
                HmiFile.Status.DeleteStep := FILE_SELECT_OLDEST_FILES_0;
            ELSIF (HmiFile.Parameters.Fifo.FifoType = FILE_FIFO_SIZE_OF_FOLDER) THEN
				HmiFile.Status.DeleteStep := FILE_CALC_FOLDER_SIZE;
            END_IF

        FILE_SELECT_OLDEST_FILES_0:
			// Scan and select all file over the filter setting
			IF (MpFileManagerUIConnect.Status = mpFILE_UI_STATUS_IDLE) THEN
				IF MpFileManagerUIConnect.File.PathInfo.FileCount > 1 THEN
           			MpFileManagerUIConnect.File.MultiSelect := TRUE;
				END_IF
				HmiFile.Status.AutoDeleteSelected := 0;
				FOR i := 0 TO ((SIZEOF(HmiFile.Status.FileNames)/SIZEOF(HmiFile.Status.FileNames[0])) - 1) DO
					IF i >= HmiFile.Parameters.Fifo.MaxNumberOfFiles THEN
						MpFileManagerUIConnect.File.List.Items[0].IsSelected := FALSE;
						IF (MpFileManagerUIConnect.File.List.Items[i].ItemType <> mpFILE_ITEM_TYPE_NONE) AND NOT MpFileManagerUIConnect.File.List.Items[i].IsFolder THEN
							MpFileManagerUIConnect.File.List.Items[i].IsSelected := TRUE;
							HmiFile.Status.AutoDeleteSelected := HmiFile.Status.AutoDeleteSelected + 1;
						END_IF
					END_IF
				END_FOR

				IF (HmiFile.Status.AutoDeleteSelected > 0) THEN
					HmiFile.Status.DeleteStep := FILE_DELETE_FILES;
				ELSE
					MpFileManagerUIConnect.File.MultiSelect := FALSE;
					HmiFile.Status.DeleteStep := FILE_RESET_SORT_BY;
				END_IF
			END_IF

		FILE_CALC_FOLDER_SIZE:
			// Calculate the overall file size in the open folder
				HmiFile.Status.FolderSize := 0;
				FOR i := 0 TO ((SIZEOF(HmiFile.Status.FileNames)/SIZEOF(HmiFile.Status.FileNames[0])) - 1) DO
					IF MpFileManagerUIConnect.File.List.Items[i].ItemType <> mpFILE_ITEM_TYPE_FOLDER THEN
						HmiFile.Status.FolderSize := HmiFile.Status.FolderSize + UDINT_TO_REAL(MpFileManagerUIConnect.File.List.Items[i].Size);
					END_IF
				END_FOR
				IF (HmiFile.Status.FolderSize > HmiFile.Parameters.Fifo.MaxFolderSize) THEN
					HmiFile.Status.DeleteStep := FILE_SELECT_OLDEST_FILES_1;
				ELSE
					HmiFile.Status.DeleteStep := FILE_RESET_SORT_BY;
				END_IF

		FILE_SELECT_OLDEST_FILES_1:
			// Scan and select all file over the filter setting
			IF (MpFileManagerUIConnect.Status = mpFILE_UI_STATUS_IDLE) THEN
				MpFileManagerUIConnect.File.List.Items[(MpFileManagerUIConnect.File.PathInfo.FileCount - 1)].IsSelected := TRUE;
				HmiFile.Status.DeleteStep := FILE_DELETE_FILES;
			END_IF

		FILE_DELETE_FILES:
			// Set command to delete the selected oldest files
			IF  (MpFileManagerUIConnect.Status = mpFILE_UI_STATUS_IDLE) THEN
				MpFileManagerUIConnect.File.Delete := TRUE;
			END_IF

			IF (MpFileManagerUIConnect.Status = mpFILE_UI_STATUS_DELETE) THEN
				HmiFile.Status.DeleteStep := FILE_CONFIRM_DELETE;
            END_IF

		FILE_CONFIRM_DELETE:
			// Confirm the file delete
            IF (MpFileManagerUIConnect.MessageBox.Type = mpFILE_MSG_CONFIRM_DELETE) THEN
                MpFileManagerUIConnect.MessageBox.Confirm := TRUE;
            ELSIF (MpFileManagerUIConnect.Status = mpFILE_UI_STATUS_IDLE) AND (MpFileManagerUIConnect.MessageBox.LayerStatus = 1) THEN
				IF (HmiFile.Parameters.Fifo.FifoType = FILE_FIFO_SIZE_OF_FOLDER) THEN
                	HmiFile.Status.DeleteStep := FILE_CALC_FOLDER_SIZE;
				ELSE
					HmiFile.Status.DeleteStep := FILE_RESET_SORT_BY;
					MpFileManagerUIConnect.File.MultiSelect := FALSE;
				END_IF
            END_IF

		FILE_RESET_SORT_BY:
			// Restore old sort order
            IF (MpFileManagerUIConnect.File.SortOrder <> HmiFile.Parameters.OldSortOrder) THEN
                MpFileManagerUIConnect.File.SortOrder := HmiFile.Parameters.OldSortOrder;
            ELSIF (MpFileManagerUIConnect.Status = mpFILE_UI_STATUS_IDLE) THEN
                MpFileManagerUIConnect.File.Refresh := TRUE;
            END_IF

            IF (MpFileManagerUIConnect.Status = mpFILE_UI_STATUS_REFRESH) THEN
                HmiFile.Status.DeleteStep := FILE_DELETE_WAIT;
				IF (MpFileManagerUIConnect.MessageBox.Type = mpFILE_MSG_BUSY) THEN
					MpFileManagerUIConnect.MessageBox.Confirm := TRUE;
				END_IF
            END_IF
	END_CASE

	TON_ScanFolder(PT := DINT_TO_TIME(HmiFile.Parameters.Fifo.ScanInterval * 60000));

END_ACTION
```

### Program Logical/Infrastructure/File/FileMgt (IEC)

#### FileMgt.st - Init, cyclic, exit code
```iecst
//***********************************************************************
// Copyright: B&R Industrial Automation GmbH
// Author: B&R Industrial Automation GmbH
// Created: Jan 1, 2022
// Description: Tasks for File management control. The File management
// handling is done in this task.
//***********************************************************************

PROGRAM _INIT

	// Inititialize mapp function block
	MpFileManagerUIConnect.DeviceList.DeviceNames[0] := 'mappRecipe';
	MpFileManagerUIConnect.DeviceList.DeviceNames[1] := 'mappAudit';
	MpFileManagerUIConnect.DeviceList.DeviceNames[2] := 'mappReport';
	MpFileManagerUIConnect.DeviceList.DeviceNames[3] := 'mappData';
	MpFileManagerUIConnect.DeviceList.DeviceNames[4] := 'mappBackup';
	MpFileManagerUIConnect.DeviceList.DeviceNames[5] := 'mappAlarmX';
	MpFileManagerUIConnect.DeviceList.DeviceNames[6] := 'mappUserX';
	MpFileManagerUI_0.Enable := TRUE;
	MpFileManagerUI_0.MpLink := ADR(gMpLinkFileManagerUIFile);
	MpFileManagerUI_0.UIConnect := ADR(MpFileManagerUIConnect);
	MpFileManagerUI_0.UISetup.FileListSize := SIZEOF(MpFileManagerUIConnect.File.List.Items) / SIZEOF(MpFileManagerUIConnect.File.List.Items[0]);
	MpFileManagerUI_0();

	// Initialize FIFO feature
    HmiFile.Parameters.Fifo.DeviceName := 'mappData';
    // MaxFolderSize is in kB
	HmiFile.Parameters.Fifo.MaxFolderSize := 20000;
    HmiFile.Parameters.Fifo.MaxNumberOfFiles := 20;
    // ScanInterval is in minutes
	HmiFile.Parameters.Fifo.ScanInterval := 60;

	HmiFile.Status.DeviceDataProvider[0] := '{"value":"mappRecipe","text":"mappRecipe"}';
	HmiFile.Status.DeviceDataProvider[1] := '{"value":"mappAudit","text":"mappAudit"}';
	HmiFile.Status.DeviceDataProvider[2] := '{"value":"mappReport","text":"mappReport"}';
	HmiFile.Status.DeviceDataProvider[3] := '{"value":"mappData","text":"mappData"}';
	HmiFile.Status.DeviceDataProvider[4] := '{"value":"mappBackup","text":"mappBackup"}';
	HmiFile.Status.DeviceDataProvider[5] := '{"value":"mappAlarmX","text":"mappAlarmX"}';
	HmiFile.Status.DeviceDataProvider[6] := '{"value":"mappUserX","text":"mappUserX"}';

END_PROGRAM

PROGRAM _CYCLIC

	// Call all actions
	FormatDeviceDataProvider;
	FileManager;
	IF HmiFile.Parameters.Fifo.Enable THEN
		FIFOOperation;
	END_IF

	// Error reset
    IF NOT MpFileManagerUI_0.Error THEN
        MpFileManagerUI_0.ErrorReset := FALSE;
    END_IF

	// Assign MpLink
	MpFileManagerUI_0.MpLink := ADR(gMpLinkFileManagerUIFile);

	// Call function block
	MpFileManagerUI_0();

END_PROGRAM

PROGRAM _EXIT

	// Disable the function blocls to unlink the MpLink
	MpFileManagerUI_0.Enable := FALSE;

	// Call function block
	MpFileManagerUI_0();

END_PROGRAM
```

#### FileMgt.typ - Local data types
```iecst
TYPE
	FileHmiInterfaceType : 	STRUCT
		Commands : FileHmiCommandsType;
		Parameters : FileHmiParametersType;
		Status : FileHmiStatusType;
	END_STRUCT;
	FileDeleteStepEnum :
		(
		FILE_DELETE_WAIT := 0,
		FILE_SCAN_FOLDER_WAIT,
		FILE_SELECT_DEVICE,
		FILE_CHECK_FOR_FILTER,
		FILE_SORT_BY_DATE,
		FILE_SELECT_OLDEST_FILES_0,
		FILE_CALC_FOLDER_SIZE,
		FILE_SELECT_OLDEST_FILES_1,
		FILE_DELETE_FILES,
		FILE_CONFIRM_DELETE,
		FILE_RESET_SORT_BY
		);
	FileFifoTypeEnum :
		(
		FILE_FIFO_NUM_OF_FILES := 0,
		FILE_FIFO_SIZE_OF_FOLDER,
		FILE_FIFO_OLDER_THAN
		);
	FileHmiCommandsType : 	STRUCT
		Delete : BOOL;
		FolderUp : BOOL;
		EnterFolder : BOOL;
		MultiSelect : BOOL;
		CheckFolder : BOOL;
	END_STRUCT;
	FileHmiParaFifoType : 	STRUCT
		Enable : BOOL;
		DeviceName : STRING[50];
		FifoType : FileFifoTypeEnum;
		ScanInterval : DINT := 60; (*[minutes]*)
		MaxFileAge : UINT := 365; (*[days] Files older than 1 year will be deleted*)
		MaxFolderSize : REAL := 1000; (*[kB] - Max size of files inside the active folder*)
		MaxNumberOfFiles : UINT := 20; (*Max number of files inside active folder*)
	END_STRUCT;
	FileHmiParametersType : 	STRUCT
		SelectedIndex : USINT;
		OldSortOrder : MpFileManagerUISortOrderEnum;
		Fifo : FileHmiParaFifoType;
	END_STRUCT;
	FileTypeEnum :
		(
		FOLDER := 0,
		FILE := 1,
		FILE_SELECTED := 2
		);
	FileHmiStatusType : 	STRUCT
		FileNames : ARRAY[0..49]OF STRING[80];
		TimeStamps : ARRAY[0..49]OF DATE_AND_TIME;
		Type : ARRAY[0..49]OF DINT;
		Size : ARRAY[0..49]OF UDINT;
		DeviceDataProvider : ARRAY[0..MAX_IDX_FILE_DEV]OF STRING[100];
		DeviceName : STRING[50];
		FileName : STRING[255];
		TableConfig : ARRAY[0..1]OF STRING[120];
		IsFolder : BOOL;
		BackButton : USINT;
		DeleteStep : FileDeleteStepEnum;
		AutoDeleteSelected : USINT;
		FolderSize : REAL;
		CurrentPage : STRING[80];
	END_STRUCT;
END_TYPE
```

#### FileMgt.var - Local variables
```iecst
(********************************************************************
 * COPYRIGHT -- Bernecker + Rainer
 ********************************************************************
 * Program: FileManagement
 * File: FileManagement.var
 * Author: Bernecker + Rainer
 * Created: December , 2020
 ********************************************************************
 * Local variables of program FileManagement
 ********************************************************************)
(*File Management Variables*)
VAR
	MpFileManagerUIConnect : MpFileManagerUIConnectType;
	MpFileManagerUI_0 : MpFileManagerUI;
	Index : USINT; (*Index to loop through file devices*)
	HmiFile : FileHmiInterfaceType;
	i : USINT;
	DeviceCount : USINT;
	FolderDepthCount : USINT;
	R_TRIG_CheckStatus : R_TRIG;
	TON_ScanFolder : TON;
END_VAR
(*Defines*)
VAR CONSTANT
	MAX_IDX_FILE_DEV : USINT := MAX_IDX_USB_DEV_LIST + 7;
END_VAR
```

#### HMIActions.st
```iecst
ACTION FormatDeviceDataProvider:

	// Select CF device if USB device is not available
    FOR Index := 0 TO MAX_IDX_USB_DEV_LIST DO
        IF gUSBAvailable[Index] THEN

            brsstrcpy(ADR(HmiFile.Status.DeviceDataProvider[Index + 7]), ADR('{"value":"USB'));
            brsitoa(Index + 1, ADR(HmiFile.Status.DeviceDataProvider[Index + 7]) + brsstrlen(ADR(HmiFile.Status.DeviceDataProvider[Index + 7])));

			brsstrcat(ADR(HmiFile.Status.DeviceDataProvider[Index + 7]), ADR('","text":"USB'));
            brsitoa(Index + 1, ADR(HmiFile.Status.DeviceDataProvider[Index + 7]) + brsstrlen(ADR(HmiFile.Status.DeviceDataProvider[Index + 7])));
            brsstrcat(ADR(HmiFile.Status.DeviceDataProvider[Index + 7]), ADR('"}'));

		    brsstrcpy(ADR(MpFileManagerUIConnect.DeviceList.DeviceNames[Index + 7]), ADR('USB'));
            brsitoa(Index + 1, ADR(MpFileManagerUIConnect.DeviceList.DeviceNames[Index + 7]) + brsstrlen(ADR(MpFileManagerUIConnect.DeviceList.DeviceNames[Index + 7])));
        ELSE
            brsmemset(ADR(HmiFile.Status.DeviceDataProvider[Index + 7]), 0, SIZEOF(HmiFile.Status.DeviceDataProvider[Index + 7]));
            brsmemset(ADR(MpFileManagerUIConnect.DeviceList.DeviceNames[Index + 7]), 0, SIZEOF(MpFileManagerUIConnect.DeviceList.DeviceNames[Index + 7]));
        END_IF
    END_FOR

	// Configure visible device list
    brsstrcpy(ADR(HmiFile.Status.TableConfig[0]), ADR('{ "specRows": [{"from":'));
	FOR i := 0 TO 9 DO
		IF MpFileManagerUIConnect.DeviceList.DeviceNames[i] <> '' THEN
			DeviceCount := i+1;
		END_IF
	END_FOR
	brsitoa((DeviceCount), ADR(HmiFile.Status.TableConfig[0]) + brsstrlen(ADR(HmiFile.Status.TableConfig[0])));
    brsstrcat(ADR(HmiFile.Status.TableConfig[0]),  ADR(',"to":9, "visible":false}]}'));

    // Configure visible file list
    brsstrcpy(ADR(HmiFile.Status.TableConfig[1]), ADR('{ "specRows": [{"from":'));
    brsitoa((MpFileManagerUIConnect.File.PathInfo.FileCount + MpFileManagerUIConnect.File.PathInfo.FolderCount), ADR(HmiFile.Status.TableConfig[1]) + brsstrlen(ADR(HmiFile.Status.TableConfig[1])));
    brsstrcat(ADR(HmiFile.Status.TableConfig[1]),  ADR(',"to":49, "visible":false}]}'));

END_ACTION

ACTION FileManager:

    MpFileManagerUI_0.MpLink := ADR(gMpLinkFileManagerUIFile);
    MpFileManagerUI_0.UIConnect := ADR(MpFileManagerUIConnect);
    MpFileManagerUI_0();
    FOR i:=0 TO ((SIZEOF(HmiFile.Status.FileNames)/SIZEOF(HmiFile.Status.FileNames[0]))-1) DO
        HmiFile.Status.FileNames[i] := MpFileManagerUIConnect.File.List.Items[i].Name;
        HmiFile.Status.TimeStamps[i] := MpFileManagerUIConnect.File.List.Items[i].LastModified;
        HmiFile.Status.Size[i] := REAL_TO_UDINT(UDINT_TO_REAL(MpFileManagerUIConnect.File.List.Items[i].Size) * 0.001);

		// Set image array based on item type
		IF MpFileManagerUIConnect.File.List.Items[i].IsFolder THEN
			HmiFile.Status.Type[i] := FOLDER;
		ELSIF NOT MpFileManagerUIConnect.File.List.Items[i].IsFolder AND MpFileManagerUIConnect.File.List.Items[i].IsSelected THEN
			HmiFile.Status.Type[i] := FILE_SELECTED;
		ELSE
			HmiFile.Status.Type[i] := FILE;
		END_IF

		// Set file selected when the table is clicked Single and MultiSelect
		IF HmiFile.Status.DeleteStep = FILE_DELETE_WAIT THEN
			IF (MpFileManagerUIConnect.File.MultiSelect = FALSE) THEN
				IF (i = HmiFile.Parameters.SelectedIndex) THEN
					MpFileManagerUIConnect.File.List.Items[i].IsSelected := TRUE;
				ELSE
					MpFileManagerUIConnect.File.List.Items[i].IsSelected := FALSE;
				END_IF
			ELSIF (MpFileManagerUIConnect.File.MultiSelect = TRUE) AND HmiFile.Commands.MultiSelect THEN
				IF (i = HmiFile.Parameters.SelectedIndex) AND NOT MpFileManagerUIConnect.File.List.Items[i].IsSelected THEN
					MpFileManagerUIConnect.File.List.Items[i].IsSelected := TRUE;
					HmiFile.Commands.MultiSelect := FALSE;
				ELSIF (i = HmiFile.Parameters.SelectedIndex) AND MpFileManagerUIConnect.File.List.Items[i].IsSelected THEN
					MpFileManagerUIConnect.File.List.Items[i].IsSelected := FALSE;
					HmiFile.Commands.MultiSelect := FALSE;
				END_IF
			END_IF
		END_IF
    END_FOR

	// Read currently selected device name for HMI
	HmiFile.Status.DeviceName := MpFileManagerUIConnect.DeviceList.DeviceNames[MpFileManagerUIConnect.DeviceList.SelectedIndex];

	// Read if current selected object is folder
	HmiFile.Status.IsFolder := MpFileManagerUIConnect.File.List.Items[HmiFile.Parameters.SelectedIndex].IsFolder;

	// Control the folder structure when entering and leaving folders
	IF (HmiFile.Commands.EnterFolder) AND MpFileManagerUIConnect.File.List.Items[HmiFile.Parameters.SelectedIndex].IsFolder THEN
		HmiFile.Commands.EnterFolder := FALSE;
		MpFileManagerUIConnect.File.EnterFolder := TRUE;
		FolderDepthCount := FolderDepthCount + 1;
	ELSE
		HmiFile.Commands.EnterFolder := FALSE;
	END_IF

	IF EDGEPOS(HmiFile.Commands.FolderUp) AND (HmiFile.Status.BackButton > 0) THEN
		HmiFile.Commands.FolderUp := FALSE;
		MpFileManagerUIConnect.File.FolderUp := TRUE;
		FolderDepthCount := FolderDepthCount - 1;
	END_IF

	IF FolderDepthCount > 0 THEN
		HmiFile.Status.BackButton := TRUE;
	ELSE
		HmiFile.Status.BackButton := FALSE;
	END_IF

END_ACTION
```
